KUKA KRL program: f1_Kuka_APT213T03S13.SRC

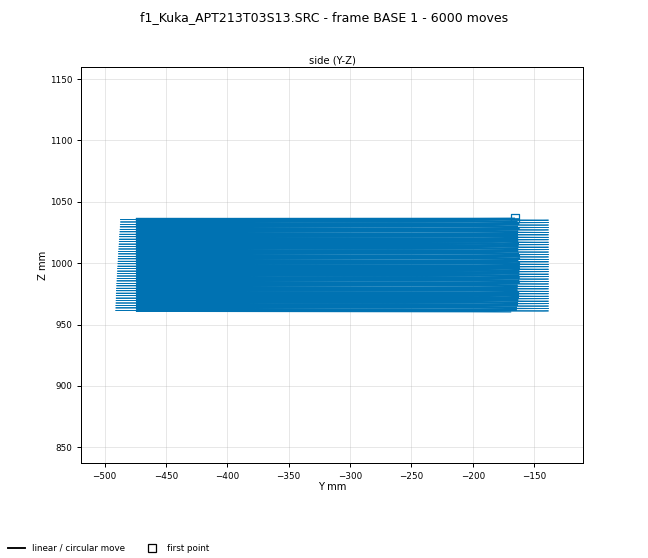
[picture p0: tool path of f1_Kuka_APT213T03S13.SRC in frame BASE 1, 6000 of 6001 moves have a stored position in this frame; points joined in program order, loops and branches not executed]
&ACCESS RVP
&REL 2
&PARAM TEMPLATE = C:\KRC\Roboter\Template\vorgabe
&PARAM EDITMASK = *
DEF f1_Kuka_APT213T03S13()


;FOLD INI;%{PE}%V3.2.0,%MKUKATPBASIS,%CINIT,%VCOMMON,%P
  ;FOLD BAS INI;%{E}%V3.2.0,%MKUKATPBASIS,%CINIT,%VINIT,%P
    GLOBAL INTERRUPT DECL 3 WHEN $STOPMESS==TRUE DO IR_STOPM ( )
    INTERRUPT ON 3
    BAS (#INITMOV,0 )
  ;ENDFOLD (BAS INI)
  ;FOLD USER INI;%{E}%V3.2.0,%MKUKATPUSER,%CINIT,%VINIT,%P
    ;Make your modifications here
  ;ENDFOLD (USER INI)
;ENDFOLD (INI)


;*** Make Null PTP Move
  PTP $pos_act

;*** Auto Load The Correct TOOL Data
  $tool=tool_data[3]

;*** Auto Load The Correct BASE Data
  $base=base_data[1]

  $ADVANCE = 5

;*** Restate Last Velocity
MMPM(30000.0)
SetRPM(6000)
LIN {X 0.063,Y -165.933,Z 1036.809,A 0.000,B 0.000,C 90.000,E1 145.515} C_DIS
LIN {X -0.044,Y -170.922,Z 1036.789,A 0.000,B 0.000,C 90.000,E1 142.065} C_DIS
LIN {X -0.018,Y -175.791,Z 1036.770,A 0.000,B 0.000,C 90.000,E1 138.609} C_DIS
LIN {X -0.018,Y -181.399,Z 1036.751,A 0.000,B 0.000,C 90.000,E1 135.202} C_DIS
LIN {X -0.014,Y -186.897,Z 1036.732,A 0.000,B 0.000,C 90.000,E1 131.838} C_DIS
LIN {X -0.063,Y -191.479,Z 1036.719,A 0.000,B 0.000,C 90.000,E1 129.358} C_DIS
LIN {X -0.019,Y -197.520,Z 1036.700,A 0.000,B 0.000,C 90.000,E1 125.964} C_DIS
LIN {X 0.097,Y -303.588,Z 1036.700,A 0.000,B 0.000,C 90.000,E1 125.931} C_DIS
LIN {X -0.058,Y -305.059,Z 1036.700,A 0.000,B 0.000,C 90.000,E1 125.931} C_DIS
LIN {X 0.134,Y -308.841,Z 1036.699,A 0.000,B 0.000,C 90.000,E1 125.724} C_DIS
LIN {X -0.104,Y -311.070,Z 1036.698,A 0.000,B 0.000,C 90.000,E1 125.598} C_DIS
LIN {X 0.033,Y -314.160,Z 1036.696,A 0.000,B 0.000,C 90.000,E1 125.231} C_DIS
LIN {X -0.057,Y -316.144,Z 1036.694,A 0.000,B 0.000,C 90.000,E1 124.945} C_DIS
LIN {X 0.113,Y -317.699,Z 1036.692,A 0.000,B 0.000,C 90.000,E1 124.612} C_DIS
LIN {X -0.083,Y -319.007,Z 1036.691,A 0.000,B 0.000,C 90.000,E1 124.326} C_DIS
LIN {X -0.008,Y -330.156,Z 1036.673,A 0.000,B 0.000,C 90.000,E1 121.131} C_DIS
LIN {X 0.067,Y -341.560,Z 1036.657,A 0.000,B 0.000,C 90.000,E1 118.309} C_DIS
LIN {X -0.156,Y -354.382,Z 1036.642,A 0.000,B 0.000,C 90.000,E1 115.591} C_DIS
LIN {X 0.094,Y -367.068,Z 1036.629,A 0.000,B 0.000,C 90.000,E1 113.153} C_DIS
LIN {X 0.194,Y -381.055,Z 1036.616,A 0.000,B 0.000,C 90.000,E1 110.791} C_DIS
LIN {X -0.133,Y -396.444,Z 1036.603,A 0.000,B 0.000,C 90.000,E1 108.544} C_DIS
LIN {X 0.173,Y -413.344,Z 1036.590,A 0.000,B 0.000,C 90.000,E1 106.260} C_DIS
LIN {X -0.136,Y -431.875,Z 1036.578,A 0.000,B 0.000,C 90.000,E1 104.120} C_DIS
LIN {X 0.111,Y -451.748,Z 1036.567,A 0.000,B 0.000,C 90.000,E1 102.007} C_DIS
LIN {X 0.212,Y -467.042,Z 1036.559,A 0.000,B 0.000,C 90.000,E1 100.546} C_DIS
LIN {X 0.229,Y -469.174,Z 1036.557,A 0.000,B 0.000,C 90.000,E1 100.310} C_DIS
LIN {X 0.077,Y -470.911,Z 1036.556,A 0.000,B 0.000,C 90.000,E1 100.074} C_DIS
LIN {X -0.158,Y -472.215,Z 1036.555,A 0.000,B 0.000,C 90.000,E1 99.849} C_DIS
LIN {X 0.023,Y -473.839,Z 1036.552,A 0.000,B 0.000,C 90.000,E1 99.321} C_DIS
LIN {X 0.135,Y -474.404,Z 1036.549,A 0.000,B 0.000,C 90.000,E1 98.803} C_DIS
LIN {X -0.211,Y -474.005,Z 1036.546,A 0.000,B 0.000,C 90.000,E1 98.341} C_DIS
LIN {X -0.017,Y -472.586,Z 1036.543,A 0.000,B 0.000,C 90.000,E1 97.814} C_DIS
LIN {X -0.220,Y -471.422,Z 1036.542,A 0.000,B 0.000,C 90.000,E1 97.587} C_DIS
LIN {X -0.100,Y -468.092,Z 1036.539,A 0.000,B 0.000,C 90.000,E1 97.068} C_DIS
LIN {X -0.038,Y -455.730,Z 1036.529,A 0.000,B 0.000,C 90.000,E1 95.277} C_DIS
LIN {X -0.181,Y -438.069,Z 1036.515,A 0.000,B 0.000,C 90.000,E1 92.694} C_DIS
LIN {X -0.168,Y -419.039,Z 1036.497,A 0.000,B 0.000,C 90.000,E1 89.484} C_DIS
LIN {X 0.171,Y -407.384,Z 1036.485,A 0.000,B 0.000,C 90.000,E1 87.249} C_DIS
LIN {X -0.201,Y -396.986,Z 1036.474,A 0.000,B 0.000,C 90.000,E1 85.355} C_DIS
LIN {X 0.031,Y -387.808,Z 1036.465,A 0.000,B 0.000,C 90.000,E1 83.628} C_DIS
LIN {X 0.138,Y -378.455,Z 1036.455,A 0.000,B 0.000,C 90.000,E1 81.894} C_DIS
LIN {X 0.131,Y -368.748,Z 1036.445,A 0.000,B 0.000,C 90.000,E1 80.151} C_DIS
LIN {X -0.087,Y -357.143,Z 1036.434,A 0.000,B 0.000,C 90.000,E1 78.117} C_DIS
LIN {X 0.011,Y -347.219,Z 1036.424,A 0.000,B 0.000,C 90.000,E1 76.297} C_DIS
LIN {X -0.112,Y -334.181,Z 1036.410,A 0.000,B 0.000,C 90.000,E1 73.866} C_DIS
LIN {X 0.058,Y -321.599,Z 1036.396,A 0.000,B 0.000,C 90.000,E1 71.329} C_DIS
LIN {X 0.143,Y -306.483,Z 1036.379,A 0.000,B 0.000,C 90.000,E1 68.103} C_DIS
LIN {X -0.076,Y -296.232,Z 1036.366,A 0.000,B 0.000,C 90.000,E1 65.845} C_DIS
LIN {X 0.120,Y -284.774,Z 1036.351,A 0.000,B 0.000,C 90.000,E1 63.127} C_DIS
LIN {X -0.163,Y -274.969,Z 1036.338,A 0.000,B 0.000,C 90.000,E1 60.795} C_DIS
LIN {X -0.094,Y -263.959,Z 1036.322,A 0.000,B 0.000,C 90.000,E1 57.995} C_DIS
LIN {X 0.116,Y -253.213,Z 1036.306,A 0.000,B 0.000,C 90.000,E1 55.102} C_DIS
LIN {X 0.128,Y -241.650,Z 1036.288,A 0.000,B 0.000,C 90.000,E1 51.823} C_DIS
LIN {X 0.082,Y -230.864,Z 1036.270,A 0.000,B 0.000,C 90.000,E1 48.485} C_DIS
LIN {X -0.075,Y -221.890,Z 1036.253,A 0.000,B 0.000,C 90.000,E1 45.486} C_DIS
LIN {X 0.039,Y -213.400,Z 1036.235,A 0.000,B 0.000,C 90.000,E1 42.366} C_DIS
LIN {X 0.129,Y -205.412,Z 1036.218,A 0.000,B 0.000,C 90.000,E1 39.197} C_DIS
LIN {X 0.081,Y -197.949,Z 1036.200,A 0.000,B 0.000,C 90.000,E1 36.011} C_DIS
LIN {X 0.101,Y -191.076,Z 1036.182,A 0.000,B 0.000,C 90.000,E1 32.752} C_DIS
LIN {X 0.069,Y -184.943,Z 1036.164,A 0.000,B 0.000,C 90.000,E1 29.461} C_DIS
LIN {X -0.060,Y -179.566,Z 1036.145,A 0.000,B 0.000,C 90.000,E1 26.155} C_DIS
LIN {X -0.062,Y -175.003,Z 1036.126,A 0.000,B 0.000,C 90.000,E1 22.770} C_DIS
LIN {X 0.014,Y -171.158,Z 1036.107,A 0.000,B 0.000,C 90.000,E1 19.322} C_DIS
LIN {X -0.003,Y -167.410,Z 1036.083,A 0.000,B 0.000,C 90.000,E1 15.009} C_DIS
LIN {X -0.019,Y -164.696,Z 1036.059,A 0.000,B 0.000,C 90.000,E1 10.658} C_DIS
LIN {X 0.058,Y -162.489,Z 1036.020,A 0.000,B 0.000,C 90.000,E1 3.612} C_DIS
LIN {X -0.061,Y -163.809,Z 1035.963,A 0.000,B 0.000,C 90.000,E1 353.394} C_DIS
LIN {X -0.005,Y -166.537,Z 1035.934,A 0.000,B 0.000,C 90.000,E1 348.117} C_DIS
LIN {X 0.070,Y -169.974,Z 1035.910,A 0.000,B 0.000,C 90.000,E1 343.740} C_DIS
LIN {X -0.022,Y -173.413,Z 1035.891,A 0.000,B 0.000,C 90.000,E1 340.315} C_DIS
LIN {X 0.038,Y -177.583,Z 1035.872,A 0.000,B 0.000,C 90.000,E1 336.869} C_DIS
LIN {X -0.075,Y -182.601,Z 1035.853,A 0.000,B 0.000,C 90.000,E1 333.512} C_DIS
LIN {X 0.025,Y -188.479,Z 1035.834,A 0.000,B 0.000,C 90.000,E1 330.127} C_DIS
LIN {X -0.025,Y -195.149,Z 1035.816,A 0.000,B 0.000,C 90.000,E1 326.834} C_DIS
LIN {X -0.029,Y -202.523,Z 1035.798,A 0.000,B 0.000,C 90.000,E1 323.577} C_DIS
LIN {X 0.034,Y -210.397,Z 1035.780,A 0.000,B 0.000,C 90.000,E1 320.356} C_DIS
LIN {X 0.035,Y -220.038,Z 1035.760,A 0.000,B 0.000,C 90.000,E1 316.824} C_DIS
LIN {X -0.120,Y -229.416,Z 1035.743,A 0.000,B 0.000,C 90.000,E1 313.785} C_DIS
LIN {X -0.158,Y -238.562,Z 1035.728,A 0.000,B 0.000,C 90.000,E1 311.148} C_DIS
LIN {X -0.114,Y -247.580,Z 1035.716,A 0.000,B 0.000,C 90.000,E1 308.910} C_DIS
LIN {X -0.070,Y -256.075,Z 1035.706,A 0.000,B 0.000,C 90.000,E1 307.076} C_DIS
LIN {X 0.008,Y -265.532,Z 1035.696,A 0.000,B 0.000,C 90.000,E1 305.264} C_DIS
LIN {X -0.056,Y -283.955,Z 1035.678,A 0.000,B 0.000,C 90.000,E1 302.133} C_DIS
LIN {X 0.043,Y -303.913,Z 1035.662,A 0.000,B 0.000,C 90.000,E1 299.077} C_DIS
LIN {X 0.026,Y -320.653,Z 1035.649,A 0.000,B 0.000,C 90.000,E1 296.796} C_DIS
LIN {X 0.026,Y -333.786,Z 1035.640,A 0.000,B 0.000,C 90.000,E1 295.207} C_DIS
LIN {X 0.005,Y -350.088,Z 1035.630,A 0.000,B 0.000,C 90.000,E1 293.462} C_DIS
LIN {X 0.000,Y -374.980,Z 1035.617,A 0.000,B 0.000,C 90.000,E1 291.099} C_DIS
LIN {X -0.066,Y -388.784,Z 1035.610,A 0.000,B 0.000,C 90.000,E1 289.885} C_DIS
LIN {X -0.057,Y -402.518,Z 1035.604,A 0.000,B 0.000,C 90.000,E1 288.671} C_DIS
LIN {X 0.025,Y -413.232,Z 1035.598,A 0.000,B 0.000,C 90.000,E1 287.692} C_DIS
LIN {X -0.064,Y -420.992,Z 1035.594,A 0.000,B 0.000,C 90.000,E1 286.968} C_DIS
LIN {X -0.093,Y -428.488,Z 1035.590,A 0.000,B 0.000,C 90.000,E1 286.205} C_DIS
LIN {X 0.073,Y -438.206,Z 1035.584,A 0.000,B 0.000,C 90.000,E1 285.134} C_DIS
LIN {X 0.162,Y -447.427,Z 1035.578,A 0.000,B 0.000,C 90.000,E1 284.064} C_DIS
LIN {X -0.004,Y -453.748,Z 1035.574,A 0.000,B 0.000,C 90.000,E1 283.300} C_DIS
LIN {X -0.110,Y -459.574,Z 1035.570,A 0.000,B 0.000,C 90.000,E1 282.535} C_DIS
LIN {X -0.173,Y -464.897,Z 1035.565,A 0.000,B 0.000,C 90.000,E1 281.771} C_DIS
LIN {X -0.187,Y -469.646,Z 1035.561,A 0.000,B 0.000,C 90.000,E1 281.007} C_DIS
LIN {X 0.212,Y -473.791,Z 1035.557,A 0.000,B 0.000,C 90.000,E1 280.197} C_DIS
LIN {X 0.195,Y -477.338,Z 1035.553,A 0.000,B 0.000,C 90.000,E1 279.443} C_DIS
LIN {X -0.268,Y -480.332,Z 1035.548,A 0.000,B 0.000,C 90.000,E1 278.746} C_DIS
LIN {X -0.047,Y -482.023,Z 1035.546,A 0.000,B 0.000,C 90.000,E1 278.219} C_DIS
LIN {X -0.190,Y -484.661,Z 1035.540,A 0.000,B 0.000,C 90.000,E1 277.239} C_DIS
LIN {X -0.007,Y -485.661,Z 1035.537,A 0.000,B 0.000,C 90.000,E1 276.720} C_DIS
LIN {X 0.186,Y -486.404,Z 1035.535,A 0.000,B 0.000,C 90.000,E1 276.201} C_DIS
LIN {X -0.101,Y -486.901,Z 1035.532,A 0.000,B 0.000,C 90.000,E1 275.739} C_DIS
LIN {X 0.100,Y -487.025,Z 1035.529,A 0.000,B 0.000,C 90.000,E1 275.220} C_DIS
LIN {X -0.183,Y -486.708,Z 1035.526,A 0.000,B 0.000,C 90.000,E1 274.759} C_DIS
LIN {X -0.019,Y -485.861,Z 1035.524,A 0.000,B 0.000,C 90.000,E1 274.245} C_DIS
LIN {X 0.180,Y -484.498,Z 1035.521,A 0.000,B 0.000,C 90.000,E1 273.726} C_DIS
LIN {X -0.141,Y -482.530,Z 1035.518,A 0.000,B 0.000,C 90.000,E1 273.269} C_DIS
LIN {X 0.204,Y -481.280,Z 1035.517,A 0.000,B 0.000,C 90.000,E1 272.980} C_DIS
LIN {X -0.129,Y -478.168,Z 1035.514,A 0.000,B 0.000,C 90.000,E1 272.522} C_DIS
LIN {X 0.002,Y -474.277,Z 1035.511,A 0.000,B 0.000,C 90.000,E1 272.007} C_DIS
LIN {X 0.126,Y -469.504,Z 1035.508,A 0.000,B 0.000,C 90.000,E1 271.489} C_DIS
LIN {X -0.108,Y -464.065,Z 1035.506,A 0.000,B 0.000,C 90.000,E1 271.031} C_DIS
LIN {X -0.020,Y -458.141,Z 1035.503,A 0.000,B 0.000,C 90.000,E1 270.573} C_DIS
LIN {X 0.113,Y -454.937,Z 1035.502,A 0.000,B 0.000,C 90.000,E1 270.344} C_DIS
LIN {X -0.132,Y -448.182,Z 1035.500,A 0.000,B 0.000,C 90.000,E1 270.000} C_DIS
LIN {X 0.097,Y -440.660,Z 1035.498,A 0.000,B 0.000,C 90.000,E1 269.656} C_DIS
LIN {X 0.026,Y -432.481,Z 1035.497,A 0.000,B 0.000,C 90.000,E1 269.427} C_DIS
LIN {X 0.074,Y -423.893,Z 1035.496,A 0.000,B 0.000,C 90.000,E1 269.255} C_DIS
LIN {X 0.081,Y -414.964,Z 1035.495,A 0.000,B 0.000,C 90.000,E1 269.141} C_DIS
LIN {X 0.181,Y -401.514,Z 1035.495,A 0.000,B 0.000,C 90.000,E1 269.026} C_DIS
LIN {X 0.067,Y -397.775,Z 1035.495,A 0.000,B 0.000,C 90.000,E1 269.026} C_DIS
LIN {X 0.005,Y -181.325,Z 1035.495,A 0.000,B 0.000,C 90.000,E1 269.026} C_DIS
LIN {X 0.010,Y -180.904,Z 1035.474,A 0.000,B 0.000,C 90.000,E1 265.298} C_DIS
LIN {X -0.041,Y -180.245,Z 1035.464,A 0.000,B 0.000,C 90.000,E1 263.628} C_DIS
LIN {X -0.021,Y -178.733,Z 1035.441,A 0.000,B 0.000,C 90.000,E1 259.398} C_DIS
LIN {X 0.046,Y -175.781,Z 1035.413,A 0.000,B 0.000,C 90.000,E1 254.283} C_DIS
LIN {X 0.033,Y -171.965,Z 1035.384,A 0.000,B 0.000,C 90.000,E1 249.156} C_DIS
LIN {X 0.071,Y -171.362,Z 1035.380,A 0.000,B 0.000,C 90.000,E1 248.284} C_DIS
LIN {X 0.048,Y -167.610,Z 1035.355,A 0.000,B 0.000,C 90.000,E1 243.973} C_DIS
LIN {X 0.060,Y -166.258,Z 1035.346,A 0.000,B 0.000,C 90.000,E1 242.231} C_DIS
LIN {X 0.048,Y -163.012,Z 1035.326,A 0.000,B 0.000,C 90.000,E1 238.742} C_DIS
LIN {X -0.040,Y -160.935,Z 1035.312,A 0.000,B 0.000,C 90.000,E1 236.135} C_DIS
LIN {X 0.071,Y -157.694,Z 1035.292,A 0.000,B 0.000,C 90.000,E1 232.557} C_DIS
LIN {X 0.008,Y -155.734,Z 1035.277,A 0.000,B 0.000,C 90.000,E1 229.908} C_DIS
LIN {X 0.062,Y -151.993,Z 1035.252,A 0.000,B 0.000,C 90.000,E1 225.405} C_DIS
LIN {X 0.078,Y -150.237,Z 1035.237,A 0.000,B 0.000,C 90.000,E1 222.690} C_DIS
LIN {X 0.001,Y -146.996,Z 1035.212,A 0.000,B 0.000,C 90.000,E1 218.177} C_DIS
LIN {X -0.009,Y -145.582,Z 1035.197,A 0.000,B 0.000,C 90.000,E1 215.438} C_DIS
LIN {X -0.015,Y -142.971,Z 1035.171,A 0.000,B 0.000,C 90.000,E1 210.846} C_DIS
LIN {X 0.038,Y -141.597,Z 1035.151,A 0.000,B 0.000,C 90.000,E1 207.129} C_DIS
LIN {X -0.046,Y -139.422,Z 1035.115,A 0.000,B 0.000,C 90.000,E1 200.663} C_DIS
LIN {X 0.005,Y -139.149,Z 1035.104,A 0.000,B 0.000,C 90.000,E1 198.779} C_DIS
LIN {X 0.027,Y -138.345,Z 1035.058,A 0.000,B 0.000,C 90.000,E1 190.366} C_DIS
LIN {X 0.013,Y -139.487,Z 1035.006,A 0.000,B 0.000,C 90.000,E1 181.031} C_DIS
LIN {X -0.047,Y -141.088,Z 1034.975,A 0.000,B 0.000,C 90.000,E1 175.469} C_DIS
LIN {X 0.048,Y -142.464,Z 1034.959,A 0.000,B 0.000,C 90.000,E1 172.648} C_DIS
LIN {X -0.004,Y -144.709,Z 1034.934,A 0.000,B 0.000,C 90.000,E1 168.049} C_DIS
LIN {X -0.053,Y -147.307,Z 1034.913,A 0.000,B 0.000,C 90.000,E1 164.393} C_DIS
LIN {X -0.038,Y -150.628,Z 1034.888,A 0.000,B 0.000,C 90.000,E1 159.826} C_DIS
LIN {X 0.039,Y -154.104,Z 1034.868,A 0.000,B 0.000,C 90.000,E1 156.177} C_DIS
LIN {X -0.038,Y -157.528,Z 1034.848,A 0.000,B 0.000,C 90.000,E1 152.615} C_DIS
LIN {X -0.093,Y -161.762,Z 1034.828,A 0.000,B 0.000,C 90.000,E1 149.076} C_DIS
LIN {X 0.012,Y -165.955,Z 1034.808,A 0.000,B 0.000,C 90.000,E1 145.515} C_DIS
LIN {X 0.008,Y -170.948,Z 1034.789,A 0.000,B 0.000,C 90.000,E1 142.029} C_DIS
LIN {X -0.071,Y -175.817,Z 1034.770,A 0.000,B 0.000,C 90.000,E1 138.609} C_DIS
LIN {X 0.056,Y -181.424,Z 1034.751,A 0.000,B 0.000,C 90.000,E1 135.162} C_DIS
LIN {X -0.069,Y -186.927,Z 1034.732,A 0.000,B 0.000,C 90.000,E1 131.838} C_DIS
LIN {X 0.004,Y -191.506,Z 1034.719,A 0.000,B 0.000,C 90.000,E1 129.322} C_DIS
LIN {X -0.039,Y -197.441,Z 1034.700,A 0.000,B 0.000,C 90.000,E1 126.011} C_DIS
LIN {X -0.113,Y -303.232,Z 1034.700,A 0.000,B 0.000,C 90.000,E1 126.011} C_DIS
LIN {X 0.026,Y -304.438,Z 1034.700,A 0.000,B 0.000,C 90.000,E1 125.964} C_DIS
LIN {X -0.118,Y -308.771,Z 1034.699,A 0.000,B 0.000,C 90.000,E1 125.804} C_DIS
LIN {X -0.014,Y -311.160,Z 1034.698,A 0.000,B 0.000,C 90.000,E1 125.598} C_DIS
LIN {X -0.056,Y -314.414,Z 1034.696,A 0.000,B 0.000,C 90.000,E1 125.231} C_DIS
LIN {X 0.063,Y -316.358,Z 1034.694,A 0.000,B 0.000,C 90.000,E1 124.898} C_DIS
LIN {X -0.076,Y -317.878,Z 1034.692,A 0.000,B 0.000,C 90.000,E1 124.612} C_DIS
LIN {X -0.205,Y -320.168,Z 1034.689,A 0.000,B 0.000,C 90.000,E1 123.992} C_DIS
LIN {X 0.082,Y -330.261,Z 1034.673,A 0.000,B 0.000,C 90.000,E1 121.082} C_DIS
LIN {X 0.033,Y -341.681,Z 1034.657,A 0.000,B 0.000,C 90.000,E1 118.281} C_DIS
LIN {X -0.037,Y -354.521,Z 1034.642,A 0.000,B 0.000,C 90.000,E1 115.540} C_DIS
LIN {X 0.034,Y -367.223,Z 1034.629,A 0.000,B 0.000,C 90.000,E1 113.131} C_DIS
LIN {X -0.013,Y -381.228,Z 1034.615,A 0.000,B 0.000,C 90.000,E1 110.791} C_DIS
LIN {X 0.031,Y -396.636,Z 1034.603,A 0.000,B 0.000,C 90.000,E1 108.489} C_DIS
LIN {X -0.042,Y -413.556,Z 1034.590,A 0.000,B 0.000,C 90.000,E1 106.260} C_DIS
LIN {X 0.063,Y -432.111,Z 1034.578,A 0.000,B 0.000,C 90.000,E1 104.064} C_DIS
LIN {X -0.102,Y -451.993,Z 1034.567,A 0.000,B 0.000,C 90.000,E1 102.007} C_DIS
LIN {X 0.005,Y -467.278,Z 1034.559,A 0.000,B 0.000,C 90.000,E1 100.546} C_DIS
LIN {X 0.023,Y -469.348,Z 1034.557,A 0.000,B 0.000,C 90.000,E1 100.310} C_DIS
LIN {X -0.129,Y -471.041,Z 1034.556,A 0.000,B 0.000,C 90.000,E1 100.074} C_DIS
LIN {X 0.102,Y -472.311,Z 1034.554,A 0.000,B 0.000,C 90.000,E1 99.792} C_DIS
LIN {X -0.184,Y -473.883,Z 1034.552,A 0.000,B 0.000,C 90.000,E1 99.321} C_DIS
LIN {X -0.071,Y -474.405,Z 1034.549,A 0.000,B 0.000,C 90.000,E1 98.803} C_DIS
LIN {X 0.121,Y -473.964,Z 1034.546,A 0.000,B 0.000,C 90.000,E1 98.276} C_DIS
LIN {X 0.246,Y -472.496,Z 1034.543,A 0.000,B 0.000,C 90.000,E1 97.757} C_DIS
LIN {X 0.042,Y -471.302,Z 1034.542,A 0.000,B 0.000,C 90.000,E1 97.530} C_DIS
LIN {X 0.161,Y -467.931,Z 1034.539,A 0.000,B 0.000,C 90.000,E1 97.011} C_DIS
LIN {X 0.214,Y -455.569,Z 1034.529,A 0.000,B 0.000,C 90.000,E1 95.220} C_DIS
LIN {X 0.059,Y -437.914,Z 1034.515,A 0.000,B 0.000,C 90.000,E1 92.636} C_DIS
LIN {X -0.059,Y -420.406,Z 1034.498,A 0.000,B 0.000,C 90.000,E1 89.714} C_DIS
LIN {X -0.098,Y -408.705,Z 1034.486,A 0.000,B 0.000,C 90.000,E1 87.535} C_DIS
LIN {X -0.031,Y -398.335,Z 1034.475,A 0.000,B 0.000,C 90.000,E1 85.584} C_DIS
LIN {X 0.173,Y -390.772,Z 1034.468,A 0.000,B 0.000,C 90.000,E1 84.147} C_DIS
LIN {X -0.069,Y -379.880,Z 1034.457,A 0.000,B 0.000,C 90.000,E1 82.186} C_DIS
LIN {X -0.053,Y -371.896,Z 1034.448,A 0.000,B 0.000,C 90.000,E1 80.735} C_DIS
LIN {X -0.200,Y -360.299,Z 1034.437,A 0.000,B 0.000,C 90.000,E1 78.701} C_DIS
LIN {X -0.103,Y -348.719,Z 1034.425,A 0.000,B 0.000,C 90.000,E1 76.589} C_DIS
LIN {X 0.139,Y -335.665,Z 1034.412,A 0.000,B 0.000,C 90.000,E1 74.102} C_DIS
LIN {X -0.070,Y -323.026,Z 1034.398,A 0.000,B 0.000,C 90.000,E1 71.638} C_DIS
LIN {X 0.062,Y -307.822,Z 1034.380,A 0.000,B 0.000,C 90.000,E1 68.411} C_DIS
LIN {X 0.030,Y -296.106,Z 1034.366,A 0.000,B 0.000,C 90.000,E1 65.793} C_DIS
LIN {X -0.041,Y -284.638,Z 1034.351,A 0.000,B 0.000,C 90.000,E1 63.127} C_DIS
LIN {X 0.052,Y -274.820,Z 1034.337,A 0.000,B 0.000,C 90.000,E1 60.717} C_DIS
LIN {X 0.114,Y -263.802,Z 1034.322,A 0.000,B 0.000,C 90.000,E1 57.916} C_DIS
LIN {X -0.013,Y -251.723,Z 1034.304,A 0.000,B 0.000,C 90.000,E1 54.736} C_DIS
LIN {X -0.027,Y -240.271,Z 1034.286,A 0.000,B 0.000,C 90.000,E1 51.457} C_DIS
LIN {X 0.042,Y -229.561,Z 1034.267,A 0.000,B 0.000,C 90.000,E1 48.081} C_DIS
LIN {X -0.059,Y -219.588,Z 1034.248,A 0.000,B 0.000,C 90.000,E1 44.676} C_DIS
LIN {X 0.015,Y -211.170,Z 1034.231,A 0.000,B 0.000,C 90.000,E1 41.553} C_DIS
LIN {X 0.054,Y -203.300,Z 1034.213,A 0.000,B 0.000,C 90.000,E1 38.382} C_DIS
LIN {X -0.001,Y -195.952,Z 1034.195,A 0.000,B 0.000,C 90.000,E1 35.185} C_DIS
LIN {X -0.024,Y -189.285,Z 1034.177,A 0.000,B 0.000,C 90.000,E1 31.926} C_DIS
LIN {X -0.031,Y -183.335,Z 1034.159,A 0.000,B 0.000,C 90.000,E1 28.615} C_DIS
LIN {X -0.112,Y -178.162,Z 1034.140,A 0.000,B 0.000,C 90.000,E1 25.283} C_DIS
LIN {X 0.018,Y -173.827,Z 1034.121,A 0.000,B 0.000,C 90.000,E1 21.844} C_DIS
LIN {X 0.004,Y -170.155,Z 1034.102,A 0.000,B 0.000,C 90.000,E1 18.417} C_DIS
LIN {X 0.072,Y -166.653,Z 1034.078,A 0.000,B 0.000,C 90.000,E1 14.064} C_DIS
LIN {X -0.027,Y -163.790,Z 1034.049,A 0.000,B 0.000,C 90.000,E1 8.859} C_DIS
LIN {X 0.038,Y -164.476,Z 1033.953,A 0.000,B 0.000,C 90.000,E1 351.602} C_DIS
LIN {X 0.046,Y -167.694,Z 1033.924,A 0.000,B 0.000,C 90.000,E1 346.353} C_DIS
LIN {X 0.088,Y -171.524,Z 1033.900,A 0.000,B 0.000,C 90.000,E1 342.000} C_DIS
LIN {X -0.016,Y -175.313,Z 1033.881,A 0.000,B 0.000,C 90.000,E1 338.592} C_DIS
LIN {X -0.003,Y -179.939,Z 1033.862,A 0.000,B 0.000,C 90.000,E1 335.177} C_DIS
LIN {X 0.105,Y -185.373,Z 1033.843,A 0.000,B 0.000,C 90.000,E1 331.769} C_DIS
LIN {X 0.045,Y -191.674,Z 1033.825,A 0.000,B 0.000,C 90.000,E1 328.456} C_DIS
LIN {X 0.014,Y -198.736,Z 1033.807,A 0.000,B 0.000,C 90.000,E1 325.182} C_DIS
LIN {X 0.060,Y -207.325,Z 1033.786,A 0.000,B 0.000,C 90.000,E1 321.537} C_DIS
LIN {X -0.062,Y -215.614,Z 1033.769,A 0.000,B 0.000,C 90.000,E1 318.405} C_DIS
LIN {X -0.094,Y -225.706,Z 1033.749,A 0.000,B 0.000,C 90.000,E1 314.919} C_DIS
LIN {X 0.064,Y -235.779,Z 1033.733,A 0.000,B 0.000,C 90.000,E1 311.838} C_DIS
LIN {X -0.088,Y -241.394,Z 1033.724,A 0.000,B 0.000,C 90.000,E1 310.378} C_DIS
LIN {X -0.144,Y -250.806,Z 1033.712,A 0.000,B 0.000,C 90.000,E1 308.177} C_DIS
LIN {X 0.158,Y -259.687,Z 1033.702,A 0.000,B 0.000,C 90.000,E1 306.297} C_DIS
LIN {X -0.005,Y -275.563,Z 1033.686,A 0.000,B 0.000,C 90.000,E1 303.499} C_DIS
LIN {X -0.001,Y -294.838,Z 1033.669,A 0.000,B 0.000,C 90.000,E1 300.413} C_DIS
LIN {X 0.016,Y -315.797,Z 1033.652,A 0.000,B 0.000,C 90.000,E1 297.436} C_DIS
LIN {X -0.083,Y -328.551,Z 1033.644,A 0.000,B 0.000,C 90.000,E1 295.848} C_DIS
LIN {X -0.081,Y -344.883,Z 1033.633,A 0.000,B 0.000,C 90.000,E1 294.027} C_DIS
LIN {X -0.141,Y -372.528,Z 1033.619,A 0.000,B 0.000,C 90.000,E1 291.354} C_DIS
LIN {X -0.141,Y -386.409,Z 1033.612,A 0.000,B 0.000,C 90.000,E1 290.120} C_DIS
LIN {X -0.109,Y -402.898,Z 1033.604,A 0.000,B 0.000,C 90.000,E1 288.652} C_DIS
LIN {X 0.214,Y -413.603,Z 1033.598,A 0.000,B 0.000,C 90.000,E1 287.638} C_DIS
LIN {X 0.134,Y -421.287,Z 1033.594,A 0.000,B 0.000,C 90.000,E1 286.913} C_DIS
LIN {X -0.017,Y -431.281,Z 1033.588,A 0.000,B 0.000,C 90.000,E1 285.898} C_DIS
LIN {X -0.225,Y -438.537,Z 1033.584,A 0.000,B 0.000,C 90.000,E1 285.134} C_DIS
LIN {X -0.138,Y -447.685,Z 1033.578,A 0.000,B 0.000,C 90.000,E1 284.064} C_DIS
LIN {X 0.136,Y -453.998,Z 1033.574,A 0.000,B 0.000,C 90.000,E1 283.244} C_DIS
LIN {X 0.035,Y -459.820,Z 1033.569,A 0.000,B 0.000,C 90.000,E1 282.479} C_DIS
LIN {X -0.023,Y -465.087,Z 1033.565,A 0.000,B 0.000,C 90.000,E1 281.715} C_DIS
LIN {X -0.033,Y -469.834,Z 1033.561,A 0.000,B 0.000,C 90.000,E1 280.950} C_DIS
LIN {X -0.096,Y -473.977,Z 1033.557,A 0.000,B 0.000,C 90.000,E1 280.197} C_DIS
LIN {X -0.114,Y -477.505,Z 1033.552,A 0.000,B 0.000,C 90.000,E1 279.443} C_DIS
LIN {X -0.030,Y -480.497,Z 1033.548,A 0.000,B 0.000,C 90.000,E1 278.681} C_DIS
LIN {X 0.121,Y -482.174,Z 1033.545,A 0.000,B 0.000,C 90.000,E1 278.163} C_DIS
LIN {X -0.194,Y -483.602,Z 1033.543,A 0.000,B 0.000,C 90.000,E1 277.701} C_DIS
LIN {X -0.018,Y -484.795,Z 1033.540,A 0.000,B 0.000,C 90.000,E1 277.182} C_DIS
LIN {X 0.168,Y -485.781,Z 1033.537,A 0.000,B 0.000,C 90.000,E1 276.663} C_DIS
LIN {X -0.123,Y -486.548,Z 1033.534,A 0.000,B 0.000,C 90.000,E1 276.201} C_DIS
LIN {X 0.075,Y -487.020,Z 1033.532,A 0.000,B 0.000,C 90.000,E1 275.682} C_DIS
LIN {X -0.207,Y -487.112,Z 1033.529,A 0.000,B 0.000,C 90.000,E1 275.220} C_DIS
LIN {X -0.005,Y -486.768,Z 1033.526,A 0.000,B 0.000,C 90.000,E1 274.702} C_DIS
LIN {X 0.159,Y -485.937,Z 1033.523,A 0.000,B 0.000,C 90.000,E1 274.188} C_DIS
LIN {X -0.125,Y -484.522,Z 1033.521,A 0.000,B 0.000,C 90.000,E1 273.726} C_DIS
LIN {X 0.039,Y -482.552,Z 1033.518,A 0.000,B 0.000,C 90.000,E1 273.212} C_DIS
LIN {X -0.098,Y -481.300,Z 1033.516,A 0.000,B 0.000,C 90.000,E1 272.980} C_DIS
LIN {X 0.049,Y -478.133,Z 1033.514,A 0.000,B 0.000,C 90.000,E1 272.465} C_DIS
LIN {X 0.179,Y -474.283,Z 1033.511,A 0.000,B 0.000,C 90.000,E1 271.949} C_DIS
LIN {X -0.168,Y -469.504,Z 1033.508,A 0.000,B 0.000,C 90.000,E1 271.489} C_DIS
LIN {X 0.065,Y -464.001,Z 1033.505,A 0.000,B 0.000,C 90.000,E1 270.974} C_DIS
LIN {X 0.137,Y -458.011,Z 1033.503,A 0.000,B 0.000,C 90.000,E1 270.516} C_DIS
LIN {X 0.170,Y -451.603,Z 1033.501,A 0.000,B 0.000,C 90.000,E1 270.115} C_DIS
LIN {X -0.192,Y -444.672,Z 1033.499,A 0.000,B 0.000,C 90.000,E1 269.828} C_DIS
LIN {X -0.044,Y -437.078,Z 1033.497,A 0.000,B 0.000,C 90.000,E1 269.542} C_DIS
LIN {X 0.163,Y -428.712,Z 1033.496,A 0.000,B 0.000,C 90.000,E1 269.312} C_DIS
LIN {X -0.036,Y -419.953,Z 1033.495,A 0.000,B 0.000,C 90.000,E1 269.198} C_DIS
LIN {X 0.076,Y -410.553,Z 1033.495,A 0.000,B 0.000,C 90.000,E1 269.083} C_DIS
LIN {X -0.040,Y -397.684,Z 1033.495,A 0.000,B 0.000,C 90.000,E1 269.026} C_DIS
LIN {X -0.044,Y -181.321,Z 1033.495,A 0.000,B 0.000,C 90.000,E1 269.026} C_DIS
LIN {X -0.039,Y -180.903,Z 1033.474,A 0.000,B 0.000,C 90.000,E1 265.298} C_DIS
LIN {X -0.089,Y -180.238,Z 1033.464,A 0.000,B 0.000,C 90.000,E1 263.628} C_DIS
LIN {X -0.069,Y -178.724,Z 1033.441,A 0.000,B 0.000,C 90.000,E1 259.398} C_DIS
LIN {X -0.001,Y -175.771,Z 1033.413,A 0.000,B 0.000,C 90.000,E1 254.283} C_DIS
LIN {X -0.013,Y -171.955,Z 1033.384,A 0.000,B 0.000,C 90.000,E1 249.156} C_DIS
LIN {X 0.024,Y -171.347,Z 1033.379,A 0.000,B 0.000,C 90.000,E1 248.284} C_DIS
LIN {X 0.002,Y -167.599,Z 1033.355,A 0.000,B 0.000,C 90.000,E1 243.973} C_DIS
LIN {X 0.014,Y -166.241,Z 1033.346,A 0.000,B 0.000,C 90.000,E1 242.231} C_DIS
LIN {X 0.002,Y -162.999,Z 1033.326,A 0.000,B 0.000,C 90.000,E1 238.742} C_DIS
LIN {X 0.049,Y -160.918,Z 1033.312,A 0.000,B 0.000,C 90.000,E1 236.087} C_DIS
LIN {X 0.027,Y -157.681,Z 1033.292,A 0.000,B 0.000,C 90.000,E1 232.557} C_DIS
LIN {X -0.035,Y -155.721,Z 1033.277,A 0.000,B 0.000,C 90.000,E1 229.908} C_DIS
LIN {X 0.019,Y -151.980,Z 1033.252,A 0.000,B 0.000,C 90.000,E1 225.405} C_DIS
LIN {X 0.036,Y -150.225,Z 1033.237,A 0.000,B 0.000,C 90.000,E1 222.690} C_DIS
LIN {X -0.042,Y -146.987,Z 1033.212,A 0.000,B 0.000,C 90.000,E1 218.177} C_DIS
LIN {X -0.051,Y -145.572,Z 1033.197,A 0.000,B 0.000,C 90.000,E1 215.438} C_DIS
LIN {X 0.067,Y -142.962,Z 1033.171,A 0.000,B 0.000,C 90.000,E1 210.797} C_DIS
LIN {X -0.003,Y -141.589,Z 1033.151,A 0.000,B 0.000,C 90.000,E1 207.129} C_DIS
LIN {X 0.043,Y -139.419,Z 1033.115,A 0.000,B 0.000,C 90.000,E1 200.610} C_DIS
LIN {X -0.036,Y -139.146,Z 1033.104,A 0.000,B 0.000,C 90.000,E1 198.779} C_DIS
LIN {X -0.013,Y -138.347,Z 1033.058,A 0.000,B 0.000,C 90.000,E1 190.366} C_DIS
LIN {X -0.028,Y -139.489,Z 1033.006,A 0.000,B 0.000,C 90.000,E1 181.031} C_DIS
LIN {X 0.052,Y -141.095,Z 1032.975,A 0.000,B 0.000,C 90.000,E1 175.412} C_DIS
LIN {X 0.006,Y -142.473,Z 1032.959,A 0.000,B 0.000,C 90.000,E1 172.648} C_DIS
LIN {X -0.046,Y -144.719,Z 1032.933,A 0.000,B 0.000,C 90.000,E1 168.049} C_DIS
LIN {X 0.047,Y -147.320,Z 1032.913,A 0.000,B 0.000,C 90.000,E1 164.338} C_DIS
LIN {X -0.029,Y -150.642,Z 1032.888,A 0.000,B 0.000,C 90.000,E1 159.806} C_DIS
LIN {X -0.006,Y -154.120,Z 1032.868,A 0.000,B 0.000,C 90.000,E1 156.177} C_DIS
LIN {X -0.082,Y -157.545,Z 1032.848,A 0.000,B 0.000,C 90.000,E1 152.615} C_DIS
LIN {X 0.083,Y -161.784,Z 1032.828,A 0.000,B 0.000,C 90.000,E1 148.997} C_DIS
LIN {X -0.034,Y -165.976,Z 1032.808,A 0.000,B 0.000,C 90.000,E1 145.515} C_DIS
LIN {X -0.038,Y -170.971,Z 1032.789,A 0.000,B 0.000,C 90.000,E1 142.029} C_DIS
LIN {X 0.013,Y -175.840,Z 1032.770,A 0.000,B 0.000,C 90.000,E1 138.566} C_DIS
LIN {X 0.008,Y -181.446,Z 1032.751,A 0.000,B 0.000,C 90.000,E1 135.162} C_DIS
LIN {X -0.119,Y -186.954,Z 1032.732,A 0.000,B 0.000,C 90.000,E1 131.838} C_DIS
LIN {X 0.003,Y -190.067,Z 1032.723,A 0.000,B 0.000,C 90.000,E1 130.135} C_DIS
LIN {X 0.116,Y -197.354,Z 1032.700,A 0.000,B 0.000,C 90.000,E1 126.011} C_DIS
LIN {X 0.118,Y -302.474,Z 1032.700,A 0.000,B 0.000,C 90.000,E1 126.011} C_DIS
LIN {X -0.010,Y -306.647,Z 1032.700,A 0.000,B 0.000,C 90.000,E1 125.931} C_DIS
LIN {X 0.074,Y -309.780,Z 1032.698,A 0.000,B 0.000,C 90.000,E1 125.724} C_DIS
LIN {X -0.128,Y -313.455,Z 1032.697,A 0.000,B 0.000,C 90.000,E1 125.391} C_DIS
LIN {X -0.086,Y -316.965,Z 1032.693,A 0.000,B 0.000,C 90.000,E1 124.818} C_DIS
LIN {X -0.029,Y -318.374,Z 1032.692,A 0.000,B 0.000,C 90.000,E1 124.485} C_DIS
LIN {X -0.143,Y -330.686,Z 1032.672,A 0.000,B 0.000,C 90.000,E1 121.003} C_DIS
LIN {X 0.112,Y -342.160,Z 1032.656,A 0.000,B 0.000,C 90.000,E1 118.153} C_DIS
LIN {X 0.056,Y -355.065,Z 1032.641,A 0.000,B 0.000,C 90.000,E1 115.412} C_DIS
LIN {X -0.002,Y -367.826,Z 1032.628,A 0.000,B 0.000,C 90.000,E1 113.025} C_DIS
LIN {X 0.111,Y -381.894,Z 1032.615,A 0.000,B 0.000,C 90.000,E1 110.663} C_DIS
LIN {X 0.173,Y -397.371,Z 1032.602,A 0.000,B 0.000,C 90.000,E1 108.362} C_DIS
LIN {X 0.117,Y -414.365,Z 1032.590,A 0.000,B 0.000,C 90.000,E1 106.134} C_DIS
LIN {X 0.139,Y -432.998,Z 1032.578,A 0.000,B 0.000,C 90.000,E1 103.953} C_DIS
LIN {X 0.124,Y -452.933,Z 1032.566,A 0.000,B 0.000,C 90.000,E1 101.883} C_DIS
LIN {X 0.196,Y -468.118,Z 1032.558,A 0.000,B 0.000,C 90.000,E1 100.433} C_DIS
LIN {X 0.146,Y -470.038,Z 1032.557,A 0.000,B 0.000,C 90.000,E1 100.197} C_DIS
LIN {X 0.096,Y -471.495,Z 1032.555,A 0.000,B 0.000,C 90.000,E1 99.962} C_DIS
LIN {X 0.193,Y -473.477,Z 1032.553,A 0.000,B 0.000,C 90.000,E1 99.443} C_DIS
LIN {X -0.092,Y -474.336,Z 1032.550,A 0.000,B 0.000,C 90.000,E1 98.973} C_DIS
LIN {X 0.028,Y -474.218,Z 1032.547,A 0.000,B 0.000,C 90.000,E1 98.454} C_DIS
LIN {X 0.155,Y -473.114,Z 1032.544,A 0.000,B 0.000,C 90.000,E1 97.936} C_DIS
LIN {X 0.015,Y -472.141,Z 1032.543,A 0.000,B 0.000,C 90.000,E1 97.701} C_DIS
LIN {X -0.124,Y -470.828,Z 1032.541,A 0.000,B 0.000,C 90.000,E1 97.466} C_DIS
LIN {X -0.068,Y -458.526,Z 1032.531,A 0.000,B 0.000,C 90.000,E1 95.682} C_DIS
LIN {X -0.054,Y -444.216,Z 1032.520,A 0.000,B 0.000,C 90.000,E1 93.612} C_DIS
LIN {X 0.188,Y -429.209,Z 1032.507,A 0.000,B 0.000,C 90.000,E1 91.203} C_DIS
LIN {X 0.117,Y -414.054,Z 1032.492,A 0.000,B 0.000,C 90.000,E1 88.511} C_DIS
LIN {X -0.122,Y -403.801,Z 1032.481,A 0.000,B 0.000,C 90.000,E1 86.617} C_DIS
LIN {X -0.158,Y -393.344,Z 1032.470,A 0.000,B 0.000,C 90.000,E1 84.666} C_DIS
LIN {X 0.035,Y -382.493,Z 1032.459,A 0.000,B 0.000,C 90.000,E1 82.648} C_DIS
LIN {X 0.094,Y -374.584,Z 1032.451,A 0.000,B 0.000,C 90.000,E1 81.197} C_DIS
LIN {X 0.031,Y -366.382,Z 1032.443,A 0.000,B 0.000,C 90.000,E1 79.746} C_DIS
LIN {X -0.162,Y -354.781,Z 1032.432,A 0.000,B 0.000,C 90.000,E1 77.701} C_DIS
LIN {X 0.154,Y -341.626,Z 1032.418,A 0.000,B 0.000,C 90.000,E1 75.227} C_DIS
LIN {X -0.009,Y -328.803,Z 1032.404,A 0.000,B 0.000,C 90.000,E1 72.779} C_DIS
LIN {X 0.032,Y -316.368,Z 1032.390,A 0.000,B 0.000,C 90.000,E1 70.242} C_DIS
LIN {X -0.018,Y -304.389,Z 1032.376,A 0.000,B 0.000,C 90.000,E1 67.667} C_DIS
LIN {X -0.006,Y -294.199,Z 1032.363,A 0.000,B 0.000,C 90.000,E1 65.357} C_DIS
LIN {X 0.004,Y -282.750,Z 1032.348,A 0.000,B 0.000,C 90.000,E1 62.666} C_DIS
LIN {X 0.058,Y -272.973,Z 1032.335,A 0.000,B 0.000,C 90.000,E1 60.255} C_DIS
LIN {X 0.072,Y -261.940,Z 1032.319,A 0.000,B 0.000,C 90.000,E1 57.454} C_DIS
LIN {X 0.016,Y -251.244,Z 1032.303,A 0.000,B 0.000,C 90.000,E1 54.609} C_DIS
LIN {X -0.022,Y -239.836,Z 1032.285,A 0.000,B 0.000,C 90.000,E1 51.331} C_DIS
LIN {X 0.031,Y -229.143,Z 1032.266,A 0.000,B 0.000,C 90.000,E1 47.957} C_DIS
LIN {X -0.012,Y -220.261,Z 1032.250,A 0.000,B 0.000,C 90.000,E1 44.919} C_DIS
LIN {X -0.079,Y -211.788,Z 1032.232,A 0.000,B 0.000,C 90.000,E1 41.838} C_DIS
LIN {X -0.026,Y -203.841,Z 1032.215,A 0.000,B 0.000,C 90.000,E1 38.669} C_DIS
LIN {X 0.049,Y -196.440,Z 1032.197,A 0.000,B 0.000,C 90.000,E1 35.438} C_DIS
LIN {X -0.072,Y -189.701,Z 1032.179,A 0.000,B 0.000,C 90.000,E1 32.212} C_DIS
LIN {X 0.027,Y -183.679,Z 1032.160,A 0.000,B 0.000,C 90.000,E1 28.871} C_DIS
LIN {X -0.049,Y -178.449,Z 1032.142,A 0.000,B 0.000,C 90.000,E1 25.540} C_DIS
LIN {X -0.073,Y -174.056,Z 1032.123,A 0.000,B 0.000,C 90.000,E1 22.153} C_DIS
LIN {X -0.078,Y -170.335,Z 1032.104,A 0.000,B 0.000,C 90.000,E1 18.725} C_DIS
LIN {X 0.045,Y -166.754,Z 1032.080,A 0.000,B 0.000,C 90.000,E1 14.356} C_DIS
LIN {X -0.026,Y -164.193,Z 1032.056,A 0.000,B 0.000,C 90.000,E1 10.018} C_DIS
LIN {X 0.009,Y -162.268,Z 1032.017,A 0.000,B 0.000,C 90.000,E1 2.980} C_DIS
LIN {X -0.067,Y -163.657,Z 1031.963,A 0.000,B 0.000,C 90.000,E1 353.394} C_DIS
LIN {X -0.017,Y -166.410,Z 1031.934,A 0.000,B 0.000,C 90.000,E1 348.117} C_DIS
LIN {X 0.054,Y -169.827,Z 1031.910,A 0.000,B 0.000,C 90.000,E1 343.740} C_DIS
LIN {X 0.016,Y -173.254,Z 1031.891,A 0.000,B 0.000,C 90.000,E1 340.296} C_DIS
LIN {X 0.013,Y -177.454,Z 1031.871,A 0.000,B 0.000,C 90.000,E1 336.869} C_DIS
LIN {X 0.060,Y -182.494,Z 1031.853,A 0.000,B 0.000,C 90.000,E1 333.461} C_DIS
LIN {X -0.006,Y -188.378,Z 1031.834,A 0.000,B 0.000,C 90.000,E1 330.127} C_DIS
LIN {X -0.061,Y -195.079,Z 1031.816,A 0.000,B 0.000,C 90.000,E1 326.834} C_DIS
LIN {X 0.053,Y -202.442,Z 1031.797,A 0.000,B 0.000,C 90.000,E1 323.543} C_DIS
LIN {X -0.118,Y -211.335,Z 1031.778,A 0.000,B 0.000,C 90.000,E1 319.989} C_DIS
LIN {X -0.107,Y -221.077,Z 1031.758,A 0.000,B 0.000,C 90.000,E1 316.458} C_DIS
LIN {X -0.084,Y -230.539,Z 1031.741,A 0.000,B 0.000,C 90.000,E1 313.380} C_DIS
LIN {X 0.088,Y -239.868,Z 1031.726,A 0.000,B 0.000,C 90.000,E1 310.701} C_DIS
LIN {X -0.026,Y -249.109,Z 1031.714,A 0.000,B 0.000,C 90.000,E1 308.508} C_DIS
LIN {X 0.086,Y -257.798,Z 1031.704,A 0.000,B 0.000,C 90.000,E1 306.664} C_DIS
LIN {X 0.028,Y -273.509,Z 1031.688,A 0.000,B 0.000,C 90.000,E1 303.833} C_DIS
LIN {X -0.026,Y -292.655,Z 1031.671,A 0.000,B 0.000,C 90.000,E1 300.747} C_DIS
LIN {X -0.080,Y -313.469,Z 1031.654,A 0.000,B 0.000,C 90.000,E1 297.769} C_DIS
LIN {X -0.064,Y -326.019,Z 1031.645,A 0.000,B 0.000,C 90.000,E1 296.155} C_DIS
LIN {X -0.091,Y -339.253,Z 1031.637,A 0.000,B 0.000,C 90.000,E1 294.643} C_DIS
LIN {X -0.161,Y -355.809,Z 1031.627,A 0.000,B 0.000,C 90.000,E1 292.950} C_DIS
LIN {X -0.025,Y -380.805,Z 1031.615,A 0.000,B 0.000,C 90.000,E1 290.610} C_DIS
LIN {X -0.033,Y -397.334,Z 1031.606,A 0.000,B 0.000,C 90.000,E1 289.141} C_DIS
LIN {X -0.091,Y -410.802,Z 1031.600,A 0.000,B 0.000,C 90.000,E1 287.946} C_DIS
LIN {X -0.147,Y -418.551,Z 1031.596,A 0.000,B 0.000,C 90.000,E1 287.221} C_DIS
LIN {X 0.091,Y -426.006,Z 1031.591,A 0.000,B 0.000,C 90.000,E1 286.441} C_DIS
LIN {X -0.205,Y -435.843,Z 1031.586,A 0.000,B 0.000,C 90.000,E1 285.426} C_DIS
LIN {X 0.071,Y -442.866,Z 1031.581,A 0.000,B 0.000,C 90.000,E1 284.592} C_DIS
LIN {X -0.138,Y -449.533,Z 1031.577,A 0.000,B 0.000,C 90.000,E1 283.828} C_DIS
LIN {X 0.161,Y -455.718,Z 1031.572,A 0.000,B 0.000,C 90.000,E1 283.008} C_DIS
LIN {X 0.070,Y -461.404,Z 1031.568,A 0.000,B 0.000,C 90.000,E1 282.243} C_DIS
LIN {X -0.131,Y -468.142,Z 1031.562,A 0.000,B 0.000,C 90.000,E1 281.243} C_DIS
LIN {X -0.205,Y -472.518,Z 1031.558,A 0.000,B 0.000,C 90.000,E1 280.489} C_DIS
LIN {X -0.161,Y -476.264,Z 1031.554,A 0.000,B 0.000,C 90.000,E1 279.726} C_DIS
LIN {X -0.035,Y -478.477,Z 1031.551,A 0.000,B 0.000,C 90.000,E1 279.208} C_DIS
LIN {X 0.109,Y -480.421,Z 1031.548,A 0.000,B 0.000,C 90.000,E1 278.690} C_DIS
LIN {X -0.144,Y -482.113,Z 1031.546,A 0.000,B 0.000,C 90.000,E1 278.219} C_DIS
LIN {X 0.019,Y -483.575,Z 1031.543,A 0.000,B 0.000,C 90.000,E1 277.701} C_DIS
LIN {X 0.195,Y -484.783,Z 1031.540,A 0.000,B 0.000,C 90.000,E1 277.182} C_DIS
LIN {X -0.102,Y -485.799,Z 1031.537,A 0.000,B 0.000,C 90.000,E1 276.720} C_DIS
LIN {X 0.091,Y -486.599,Z 1031.535,A 0.000,B 0.000,C 90.000,E1 276.201} C_DIS
LIN {X -0.195,Y -487.098,Z 1031.532,A 0.000,B 0.000,C 90.000,E1 275.739} C_DIS
LIN {X 0.006,Y -487.226,Z 1031.529,A 0.000,B 0.000,C 90.000,E1 275.220} C_DIS
LIN {X 0.209,Y -486.918,Z 1031.526,A 0.000,B 0.000,C 90.000,E1 274.702} C_DIS
LIN {X -0.110,Y -486.136,Z 1031.524,A 0.000,B 0.000,C 90.000,E1 274.245} C_DIS
LIN {X 0.091,Y -484.769,Z 1031.521,A 0.000,B 0.000,C 90.000,E1 273.726} C_DIS
LIN {X -0.229,Y -482.840,Z 1031.518,A 0.000,B 0.000,C 90.000,E1 273.269} C_DIS
LIN {X 0.117,Y -481.646,Z 1031.517,A 0.000,B 0.000,C 90.000,E1 272.980} C_DIS
LIN {X -0.213,Y -478.640,Z 1031.514,A 0.000,B 0.000,C 90.000,E1 272.522} C_DIS
LIN {X -0.079,Y -474.808,Z 1031.511,A 0.000,B 0.000,C 90.000,E1 272.007} C_DIS
LIN {X 0.049,Y -470.150,Z 1031.508,A 0.000,B 0.000,C 90.000,E1 271.489} C_DIS
LIN {X -0.213,Y -464.678,Z 1031.506,A 0.000,B 0.000,C 90.000,E1 271.031} C_DIS
LIN {X 0.171,Y -461.729,Z 1031.504,A 0.000,B 0.000,C 90.000,E1 270.745} C_DIS
LIN {X -0.091,Y -455.353,Z 1031.502,A 0.000,B 0.000,C 90.000,E1 270.344} C_DIS
LIN {X 0.147,Y -448.638,Z 1031.500,A 0.000,B 0.000,C 90.000,E1 269.943} C_DIS
LIN {X -0.014,Y -441.321,Z 1031.498,A 0.000,B 0.000,C 90.000,E1 269.656} C_DIS
LIN {X -0.085,Y -433.338,Z 1031.497,A 0.000,B 0.000,C 90.000,E1 269.427} C_DIS
LIN {X -0.087,Y -424.510,Z 1031.496,A 0.000,B 0.000,C 90.000,E1 269.255} C_DIS
LIN {X -0.089,Y -415.613,Z 1031.495,A 0.000,B 0.000,C 90.000,E1 269.141} C_DIS
LIN {X 0.126,Y -405.608,Z 1031.495,A 0.000,B 0.000,C 90.000,E1 269.026} C_DIS
LIN {X -0.166,Y -394.972,Z 1031.495,A 0.000,B 0.000,C 90.000,E1 269.026} C_DIS
LIN {X 0.078,Y -181.317,Z 1031.494,A 0.000,B 0.000,C 90.000,E1 268.969} C_DIS
LIN {X -0.075,Y -180.902,Z 1031.474,A 0.000,B 0.000,C 90.000,E1 265.298} C_DIS
LIN {X 0.055,Y -180.233,Z 1031.464,A 0.000,B 0.000,C 90.000,E1 263.571} C_DIS
LIN {X 0.070,Y -178.716,Z 1031.441,A 0.000,B 0.000,C 90.000,E1 259.342} C_DIS
LIN {X -0.036,Y -175.765,Z 1031.413,A 0.000,B 0.000,C 90.000,E1 254.283} C_DIS
LIN {X 0.013,Y -171.948,Z 1031.384,A 0.000,B 0.000,C 90.000,E1 249.135} C_DIS
LIN {X -0.011,Y -171.336,Z 1031.379,A 0.000,B 0.000,C 90.000,E1 248.284} C_DIS
LIN {X -0.032,Y -167.590,Z 1031.355,A 0.000,B 0.000,C 90.000,E1 243.973} C_DIS
LIN {X -0.020,Y -166.228,Z 1031.346,A 0.000,B 0.000,C 90.000,E1 242.231} C_DIS
LIN {X -0.032,Y -162.989,Z 1031.326,A 0.000,B 0.000,C 90.000,E1 238.742} C_DIS
LIN {X 0.015,Y -160.906,Z 1031.312,A 0.000,B 0.000,C 90.000,E1 236.087} C_DIS
LIN {X -0.007,Y -157.672,Z 1031.292,A 0.000,B 0.000,C 90.000,E1 232.557} C_DIS
LIN {X -0.068,Y -155.710,Z 1031.277,A 0.000,B 0.000,C 90.000,E1 229.908} C_DIS
LIN {X -0.013,Y -151.972,Z 1031.252,A 0.000,B 0.000,C 90.000,E1 225.405} C_DIS
LIN {X 0.003,Y -150.215,Z 1031.237,A 0.000,B 0.000,C 90.000,E1 222.690} C_DIS
LIN {X -0.073,Y -146.980,Z 1031.212,A 0.000,B 0.000,C 90.000,E1 218.177} C_DIS
LIN {X 0.036,Y -145.566,Z 1031.197,A 0.000,B 0.000,C 90.000,E1 215.391} C_DIS
LIN {X 0.035,Y -142.957,Z 1031.171,A 0.000,B 0.000,C 90.000,E1 210.797} C_DIS
LIN {X -0.034,Y -141.583,Z 1031.151,A 0.000,B 0.000,C 90.000,E1 207.129} C_DIS
LIN {X 0.013,Y -139.417,Z 1031.115,A 0.000,B 0.000,C 90.000,E1 200.610} C_DIS
LIN {X 0.066,Y -139.142,Z 1031.104,A 0.000,B 0.000,C 90.000,E1 198.725} C_DIS
LIN {X -0.044,Y -138.347,Z 1031.057,A 0.000,B 0.000,C 90.000,E1 190.366} C_DIS
LIN {X -0.059,Y -139.491,Z 1031.006,A 0.000,B 0.000,C 90.000,E1 181.031} C_DIS
LIN {X 0.022,Y -141.099,Z 1030.975,A 0.000,B 0.000,C 90.000,E1 175.412} C_DIS
LIN {X -0.025,Y -142.479,Z 1030.959,A 0.000,B 0.000,C 90.000,E1 172.648} C_DIS
LIN {X 0.063,Y -144.727,Z 1030.933,A 0.000,B 0.000,C 90.000,E1 167.993} C_DIS
LIN {X 0.014,Y -147.330,Z 1030.913,A 0.000,B 0.000,C 90.000,E1 164.338} C_DIS
LIN {X 0.080,Y -150.653,Z 1030.888,A 0.000,B 0.000,C 90.000,E1 159.752} C_DIS
LIN {X -0.038,Y -154.131,Z 1030.868,A 0.000,B 0.000,C 90.000,E1 156.177} C_DIS
LIN {X 0.024,Y -157.558,Z 1030.848,A 0.000,B 0.000,C 90.000,E1 152.564} C_DIS
LIN {X 0.049,Y -161.799,Z 1030.828,A 0.000,B 0.000,C 90.000,E1 148.997} C_DIS
LIN {X 0.068,Y -165.992,Z 1030.808,A 0.000,B 0.000,C 90.000,E1 145.468} C_DIS
LIN {X 0.062,Y -170.988,Z 1030.789,A 0.000,B 0.000,C 90.000,E1 141.984} C_DIS
LIN {X -0.023,Y -175.859,Z 1030.770,A 0.000,B 0.000,C 90.000,E1 138.566} C_DIS
LIN {X -0.029,Y -181.463,Z 1030.751,A 0.000,B 0.000,C 90.000,E1 135.162} C_DIS
LIN {X 0.108,Y -186.974,Z 1030.732,A 0.000,B 0.000,C 90.000,E1 131.757} C_DIS
LIN {X 0.110,Y -190.089,Z 1030.723,A 0.000,B 0.000,C 90.000,E1 130.092} C_DIS
LIN {X -0.051,Y -197.293,Z 1030.700,A 0.000,B 0.000,C 90.000,E1 126.091} C_DIS
LIN {X -0.113,Y -302.837,Z 1030.700,A 0.000,B 0.000,C 90.000,E1 126.091} C_DIS
LIN {X -0.002,Y -305.462,Z 1030.700,A 0.000,B 0.000,C 90.000,E1 126.011} C_DIS
LIN {X -0.012,Y -308.661,Z 1030.699,A 0.000,B 0.000,C 90.000,E1 125.851} C_DIS
LIN {X 0.099,Y -312.223,Z 1030.697,A 0.000,B 0.000,C 90.000,E1 125.518} C_DIS
LIN {X 0.022,Y -315.832,Z 1030.695,A 0.000,B 0.000,C 90.000,E1 125.025} C_DIS
LIN {X 0.076,Y -317.455,Z 1030.693,A 0.000,B 0.000,C 90.000,E1 124.692} C_DIS
LIN {X -0.062,Y -319.782,Z 1030.689,A 0.000,B 0.000,C 90.000,E1 124.072} C_DIS
LIN {X 0.050,Y -331.026,Z 1030.672,A 0.000,B 0.000,C 90.000,E1 120.875} C_DIS
LIN {X -0.144,Y -342.547,Z 1030.656,A 0.000,B 0.000,C 90.000,E1 118.103} C_DIS
LIN {X -0.034,Y -355.498,Z 1030.641,A 0.000,B 0.000,C 90.000,E1 115.335} C_DIS
LIN {X -0.091,Y -368.306,Z 1030.627,A 0.000,B 0.000,C 90.000,E1 112.950} C_DIS
LIN {X -0.113,Y -382.425,Z 1030.614,A 0.000,B 0.000,C 90.000,E1 110.610} C_DIS
LIN {X -0.040,Y -397.955,Z 1030.602,A 0.000,B 0.000,C 90.000,E1 108.308} C_DIS
LIN {X -0.085,Y -415.009,Z 1030.589,A 0.000,B 0.000,C 90.000,E1 106.079} C_DIS
LIN {X 0.052,Y -433.707,Z 1030.577,A 0.000,B 0.000,C 90.000,E1 103.883} C_DIS
LIN {X -0.011,Y -453.653,Z 1030.566,A 0.000,B 0.000,C 90.000,E1 101.827} C_DIS
LIN {X 0.146,Y -466.427,Z 1030.559,A 0.000,B 0.000,C 90.000,E1 100.602} C_DIS
LIN {X 0.178,Y -468.696,Z 1030.558,A 0.000,B 0.000,C 90.000,E1 100.366} C_DIS
LIN {X 0.126,Y -470.408,Z 1030.556,A 0.000,B 0.000,C 90.000,E1 100.141} C_DIS
LIN {X -0.021,Y -471.832,Z 1030.555,A 0.000,B 0.000,C 90.000,E1 99.905} C_DIS
LIN {X -0.170,Y -472.893,Z 1030.554,A 0.000,B 0.000,C 90.000,E1 99.670} C_DIS
LIN {X -0.062,Y -474.131,Z 1030.551,A 0.000,B 0.000,C 90.000,E1 99.151} C_DIS
LIN {X 0.127,Y -474.364,Z 1030.548,A 0.000,B 0.000,C 90.000,E1 98.624} C_DIS
LIN {X -0.219,Y -473.630,Z 1030.545,A 0.000,B 0.000,C 90.000,E1 98.163} C_DIS
LIN {X -0.091,Y -471.815,Z 1030.542,A 0.000,B 0.000,C 90.000,E1 97.644} C_DIS
LIN {X 0.234,Y -470.397,Z 1030.541,A 0.000,B 0.000,C 90.000,E1 97.352} C_DIS
LIN {X -0.174,Y -458.074,Z 1030.531,A 0.000,B 0.000,C 90.000,E1 95.625} C_DIS
LIN {X 0.020,Y -442.018,Z 1030.518,A 0.000,B 0.000,C 90.000,E1 93.269} C_DIS
LIN {X 0.206,Y -427.192,Z 1030.505,A 0.000,B 0.000,C 90.000,E1 90.859} C_DIS
LIN {X 0.175,Y -410.765,Z 1030.488,A 0.000,B 0.000,C 90.000,E1 87.879} C_DIS
LIN {X -0.199,Y -401.905,Z 1030.479,A 0.000,B 0.000,C 90.000,E1 86.274} C_DIS
LIN {X 0.090,Y -392.929,Z 1030.470,A 0.000,B 0.000,C 90.000,E1 84.552} C_DIS
LIN {X -0.109,Y -382.080,Z 1030.459,A 0.000,B 0.000,C 90.000,E1 82.591} C_DIS
LIN {X -0.059,Y -374.157,Z 1030.451,A 0.000,B 0.000,C 90.000,E1 81.141} C_DIS
LIN {X -0.122,Y -365.944,Z 1030.443,A 0.000,B 0.000,C 90.000,E1 79.690} C_DIS
LIN {X 0.020,Y -354.329,Z 1030.431,A 0.000,B 0.000,C 90.000,E1 77.589} C_DIS
LIN {X -0.018,Y -341.174,Z 1030.418,A 0.000,B 0.000,C 90.000,E1 75.172} C_DIS
LIN {X 0.124,Y -328.394,Z 1030.404,A 0.000,B 0.000,C 90.000,E1 72.670} C_DIS
LIN {X 0.077,Y -314.470,Z 1030.388,A 0.000,B 0.000,C 90.000,E1 69.826} C_DIS
LIN {X 0.088,Y -302.542,Z 1030.374,A 0.000,B 0.000,C 90.000,E1 67.230} C_DIS
LIN {X -0.079,Y -293.810,Z 1030.363,A 0.000,B 0.000,C 90.000,E1 65.281} C_DIS
LIN {X 0.051,Y -282.373,Z 1030.348,A 0.000,B 0.000,C 90.000,E1 62.564} C_DIS
LIN {X -0.156,Y -272.593,Z 1030.334,A 0.000,B 0.000,C 90.000,E1 60.205} C_DIS
LIN {X -0.009,Y -261.551,Z 1030.319,A 0.000,B 0.000,C 90.000,E1 57.375} C_DIS
LIN {X 0.137,Y -250.845,Z 1030.303,A 0.000,B 0.000,C 90.000,E1 54.482} C_DIS
LIN {X -0.106,Y -239.479,Z 1030.285,A 0.000,B 0.000,C 90.000,E1 51.251} C_DIS
LIN {X -0.061,Y -228.790,Z 1030.266,A 0.000,B 0.000,C 90.000,E1 47.877} C_DIS
LIN {X -0.030,Y -218.858,Z 1030.247,A 0.000,B 0.000,C 90.000,E1 44.433} C_DIS
LIN {X 0.024,Y -210.403,Z 1030.229,A 0.000,B 0.000,C 90.000,E1 41.310} C_DIS
LIN {X -0.087,Y -202.533,Z 1030.212,A 0.000,B 0.000,C 90.000,E1 38.177} C_DIS
LIN {X -0.039,Y -195.209,Z 1030.194,A 0.000,B 0.000,C 90.000,E1 34.945} C_DIS
LIN {X -0.028,Y -188.569,Z 1030.176,A 0.000,B 0.000,C 90.000,E1 31.671} C_DIS
LIN {X -0.048,Y -182.677,Z 1030.157,A 0.000,B 0.000,C 90.000,E1 28.359} C_DIS
LIN {X 0.016,Y -177.592,Z 1030.139,A 0.000,B 0.000,C 90.000,E1 24.975} C_DIS
LIN {X -0.030,Y -173.316,Z 1030.120,A 0.000,B 0.000,C 90.000,E1 21.589} C_DIS
LIN {X 0.049,Y -169.724,Z 1030.101,A 0.000,B 0.000,C 90.000,E1 18.127} C_DIS
LIN {X -0.053,Y -166.278,Z 1030.077,A 0.000,B 0.000,C 90.000,E1 13.828} C_DIS
LIN {X -0.004,Y -163.507,Z 1030.048,A 0.000,B 0.000,C 90.000,E1 8.568} C_DIS
LIN {X 0.030,Y -164.338,Z 1029.953,A 0.000,B 0.000,C 90.000,E1 351.602} C_DIS
LIN {X 0.033,Y -167.596,Z 1029.924,A 0.000,B 0.000,C 90.000,E1 346.353} C_DIS
LIN {X 0.071,Y -171.374,Z 1029.900,A 0.000,B 0.000,C 90.000,E1 342.000} C_DIS
LIN {X -0.038,Y -175.191,Z 1029.881,A 0.000,B 0.000,C 90.000,E1 338.592} C_DIS
LIN {X -0.028,Y -179.829,Z 1029.862,A 0.000,B 0.000,C 90.000,E1 335.177} C_DIS
LIN {X 0.077,Y -185.291,Z 1029.843,A 0.000,B 0.000,C 90.000,E1 331.769} C_DIS
LIN {X 0.015,Y -191.608,Z 1029.825,A 0.000,B 0.000,C 90.000,E1 328.456} C_DIS
LIN {X -0.019,Y -198.663,Z 1029.807,A 0.000,B 0.000,C 90.000,E1 325.182} C_DIS
LIN {X -0.021,Y -206.275,Z 1029.789,A 0.000,B 0.000,C 90.000,E1 321.949} C_DIS
LIN {X -0.013,Y -214.471,Z 1029.771,A 0.000,B 0.000,C 90.000,E1 318.771} C_DIS
LIN {X 0.093,Y -224.438,Z 1029.751,A 0.000,B 0.000,C 90.000,E1 315.243} C_DIS
LIN {X 0.053,Y -234.332,Z 1029.734,A 0.000,B 0.000,C 90.000,E1 312.204} C_DIS
LIN {X 0.036,Y -241.291,Z 1029.724,A 0.000,B 0.000,C 90.000,E1 310.334} C_DIS
LIN {X 0.143,Y -250.719,Z 1029.712,A 0.000,B 0.000,C 90.000,E1 308.096} C_DIS
LIN {X 0.090,Y -259.645,Z 1029.702,A 0.000,B 0.000,C 90.000,E1 306.297} C_DIS
LIN {X -0.077,Y -275.559,Z 1029.686,A 0.000,B 0.000,C 90.000,E1 303.499} C_DIS
LIN {X 0.071,Y -294.907,Z 1029.669,A 0.000,B 0.000,C 90.000,E1 300.384} C_DIS
LIN {X -0.065,Y -315.969,Z 1029.652,A 0.000,B 0.000,C 90.000,E1 297.436} C_DIS
LIN {X -0.162,Y -328.804,Z 1029.643,A 0.000,B 0.000,C 90.000,E1 295.848} C_DIS
LIN {X 0.002,Y -347.492,Z 1029.632,A 0.000,B 0.000,C 90.000,E1 293.770} C_DIS
LIN {X -0.118,Y -369.392,Z 1029.620,A 0.000,B 0.000,C 90.000,E1 291.663} C_DIS
LIN {X -0.123,Y -385.998,Z 1029.612,A 0.000,B 0.000,C 90.000,E1 290.174} C_DIS
LIN {X 0.138,Y -402.450,Z 1029.604,A 0.000,B 0.000,C 90.000,E1 288.671} C_DIS
LIN {X 0.240,Y -413.055,Z 1029.599,A 0.000,B 0.000,C 90.000,E1 287.692} C_DIS
LIN {X 0.042,Y -420.710,Z 1029.594,A 0.000,B 0.000,C 90.000,E1 286.985} C_DIS
LIN {X 0.096,Y -428.250,Z 1029.590,A 0.000,B 0.000,C 90.000,E1 286.205} C_DIS
LIN {X 0.176,Y -437.990,Z 1029.584,A 0.000,B 0.000,C 90.000,E1 285.134} C_DIS
LIN {X -0.170,Y -447.097,Z 1029.578,A 0.000,B 0.000,C 90.000,E1 284.120} C_DIS
LIN {X 0.097,Y -453.463,Z 1029.574,A 0.000,B 0.000,C 90.000,E1 283.300} C_DIS
LIN {X -0.010,Y -459.363,Z 1029.570,A 0.000,B 0.000,C 90.000,E1 282.535} C_DIS
LIN {X -0.074,Y -464.690,Z 1029.565,A 0.000,B 0.000,C 90.000,E1 281.771} C_DIS
LIN {X -0.089,Y -469.496,Z 1029.561,A 0.000,B 0.000,C 90.000,E1 281.007} C_DIS
LIN {X -0.157,Y -473.712,Z 1029.557,A 0.000,B 0.000,C 90.000,E1 280.254} C_DIS
LIN {X -0.180,Y -477.311,Z 1029.553,A 0.000,B 0.000,C 90.000,E1 279.500} C_DIS
LIN {X -0.171,Y -480.366,Z 1029.548,A 0.000,B 0.000,C 90.000,E1 278.746} C_DIS
LIN {X 0.051,Y -482.090,Z 1029.546,A 0.000,B 0.000,C 90.000,E1 278.219} C_DIS
LIN {X 0.214,Y -483.568,Z 1029.543,A 0.000,B 0.000,C 90.000,E1 277.701} C_DIS
LIN {X -0.091,Y -484.798,Z 1029.540,A 0.000,B 0.000,C 90.000,E1 277.239} C_DIS
LIN {X 0.094,Y -485.834,Z 1029.537,A 0.000,B 0.000,C 90.000,E1 276.720} C_DIS
LIN {X -0.197,Y -486.647,Z 1029.535,A 0.000,B 0.000,C 90.000,E1 276.258} C_DIS
LIN {X 0.002,Y -487.169,Z 1029.532,A 0.000,B 0.000,C 90.000,E1 275.739} C_DIS
LIN {X 0.204,Y -487.337,Z 1029.529,A 0.000,B 0.000,C 90.000,E1 275.220} C_DIS
LIN {X -0.079,Y -487.068,Z 1029.526,A 0.000,B 0.000,C 90.000,E1 274.759} C_DIS
LIN {X 0.087,Y -486.308,Z 1029.524,A 0.000,B 0.000,C 90.000,E1 274.245} C_DIS
LIN {X -0.196,Y -485.035,Z 1029.521,A 0.000,B 0.000,C 90.000,E1 273.784} C_DIS
LIN {X -0.030,Y -483.149,Z 1029.518,A 0.000,B 0.000,C 90.000,E1 273.269} C_DIS
LIN {X 0.154,Y -480.614,Z 1029.515,A 0.000,B 0.000,C 90.000,E1 272.751} C_DIS
LIN {X -0.182,Y -477.321,Z 1029.513,A 0.000,B 0.000,C 90.000,E1 272.293} C_DIS
LIN {X -0.038,Y -473.118,Z 1029.510,A 0.000,B 0.000,C 90.000,E1 271.776} C_DIS
LIN {X 0.160,Y -468.237,Z 1029.507,A 0.000,B 0.000,C 90.000,E1 271.260} C_DIS
LIN {X -0.061,Y -462.452,Z 1029.504,A 0.000,B 0.000,C 90.000,E1 270.802} C_DIS
LIN {X 0.138,Y -456.263,Z 1029.502,A 0.000,B 0.000,C 90.000,E1 270.344} C_DIS
LIN {X -0.126,Y -449.559,Z 1029.500,A 0.000,B 0.000,C 90.000,E1 270.000} C_DIS
LIN {X 0.112,Y -442.240,Z 1029.498,A 0.000,B 0.000,C 90.000,E1 269.656} C_DIS
LIN {X -0.001,Y -434.477,Z 1029.497,A 0.000,B 0.000,C 90.000,E1 269.427} C_DIS
LIN {X -0.079,Y -425.560,Z 1029.496,A 0.000,B 0.000,C 90.000,E1 269.255} C_DIS
LIN {X -0.113,Y -416.925,Z 1029.495,A 0.000,B 0.000,C 90.000,E1 269.141} C_DIS
LIN {X 0.072,Y -406.569,Z 1029.495,A 0.000,B 0.000,C 90.000,E1 269.026} C_DIS
LIN {X 0.171,Y -398.217,Z 1029.494,A 0.000,B 0.000,C 90.000,E1 268.969} C_DIS
LIN {X 0.050,Y -181.315,Z 1029.494,A 0.000,B 0.000,C 90.000,E1 268.969} C_DIS
LIN {X 0.076,Y -180.901,Z 1029.474,A 0.000,B 0.000,C 90.000,E1 265.241} C_DIS
LIN {X 0.026,Y -180.228,Z 1029.464,A 0.000,B 0.000,C 90.000,E1 263.571} C_DIS
LIN {X -0.021,Y -179.041,Z 1029.446,A 0.000,B 0.000,C 90.000,E1 260.208} C_DIS
LIN {X 0.042,Y -178.711,Z 1029.441,A 0.000,B 0.000,C 90.000,E1 259.342} C_DIS
LIN {X -0.065,Y -175.759,Z 1029.413,A 0.000,B 0.000,C 90.000,E1 254.283} C_DIS
LIN {X -0.016,Y -171.943,Z 1029.384,A 0.000,B 0.000,C 90.000,E1 249.135} C_DIS
LIN {X -0.039,Y -171.327,Z 1029.379,A 0.000,B 0.000,C 90.000,E1 248.284} C_DIS
LIN {X 0.014,Y -167.584,Z 1029.355,A 0.000,B 0.000,C 90.000,E1 243.948} C_DIS
LIN {X -0.048,Y -166.218,Z 1029.346,A 0.000,B 0.000,C 90.000,E1 242.231} C_DIS
LIN {X -0.059,Y -162.981,Z 1029.326,A 0.000,B 0.000,C 90.000,E1 238.742} C_DIS
LIN {X -0.012,Y -160.896,Z 1029.312,A 0.000,B 0.000,C 90.000,E1 236.087} C_DIS
LIN {X -0.033,Y -157.664,Z 1029.292,A 0.000,B 0.000,C 90.000,E1 232.557} C_DIS
LIN {X -0.095,Y -155.703,Z 1029.277,A 0.000,B 0.000,C 90.000,E1 229.908} C_DIS
LIN {X -0.039,Y -151.965,Z 1029.252,A 0.000,B 0.000,C 90.000,E1 225.405} C_DIS
LIN {X -0.023,Y -150.207,Z 1029.237,A 0.000,B 0.000,C 90.000,E1 222.690} C_DIS
LIN {X -0.008,Y -146.974,Z 1029.212,A 0.000,B 0.000,C 90.000,E1 218.141} C_DIS
LIN {X 0.011,Y -145.560,Z 1029.197,A 0.000,B 0.000,C 90.000,E1 215.391} C_DIS
LIN {X 0.009,Y -142.953,Z 1029.171,A 0.000,B 0.000,C 90.000,E1 210.797} C_DIS
LIN {X -0.059,Y -141.578,Z 1029.151,A 0.000,B 0.000,C 90.000,E1 207.129} C_DIS
LIN {X -0.012,Y -139.415,Z 1029.115,A 0.000,B 0.000,C 90.000,E1 200.610} C_DIS
LIN {X 0.040,Y -139.139,Z 1029.104,A 0.000,B 0.000,C 90.000,E1 198.725} C_DIS
LIN {X 0.067,Y -138.348,Z 1029.057,A 0.000,B 0.000,C 90.000,E1 190.310} C_DIS
LIN {X 0.055,Y -139.492,Z 1029.005,A 0.000,B 0.000,C 90.000,E1 180.974} C_DIS
LIN {X -0.004,Y -141.104,Z 1028.974,A 0.000,B 0.000,C 90.000,E1 175.412} C_DIS
LIN {X -0.051,Y -142.483,Z 1028.959,A 0.000,B 0.000,C 90.000,E1 172.648} C_DIS
LIN {X 0.038,Y -144.733,Z 1028.933,A 0.000,B 0.000,C 90.000,E1 167.993} C_DIS
LIN {X -0.011,Y -147.337,Z 1028.913,A 0.000,B 0.000,C 90.000,E1 164.338} C_DIS
LIN {X 0.054,Y -150.661,Z 1028.888,A 0.000,B 0.000,C 90.000,E1 159.752} C_DIS
LIN {X -0.065,Y -154.139,Z 1028.868,A 0.000,B 0.000,C 90.000,E1 156.177} C_DIS
LIN {X -0.003,Y -157.568,Z 1028.848,A 0.000,B 0.000,C 90.000,E1 152.564} C_DIS
LIN {X 0.022,Y -161.812,Z 1028.828,A 0.000,B 0.000,C 90.000,E1 148.997} C_DIS
LIN {X 0.041,Y -166.004,Z 1028.808,A 0.000,B 0.000,C 90.000,E1 145.468} C_DIS
LIN {X 0.034,Y -171.003,Z 1028.789,A 0.000,B 0.000,C 90.000,E1 141.984} C_DIS
LIN {X -0.051,Y -175.873,Z 1028.770,A 0.000,B 0.000,C 90.000,E1 138.566} C_DIS
LIN {X -0.059,Y -181.477,Z 1028.751,A 0.000,B 0.000,C 90.000,E1 135.162} C_DIS
LIN {X 0.078,Y -186.991,Z 1028.732,A 0.000,B 0.000,C 90.000,E1 131.757} C_DIS
LIN {X 0.080,Y -190.107,Z 1028.723,A 0.000,B 0.000,C 90.000,E1 130.092} C_DIS
LIN {X 0.090,Y -197.213,Z 1028.701,A 0.000,B 0.000,C 90.000,E1 126.091} C_DIS
LIN {X 0.104,Y -302.385,Z 1028.701,A 0.000,B 0.000,C 90.000,E1 126.091} C_DIS
LIN {X -0.049,Y -306.500,Z 1028.700,A 0.000,B 0.000,C 90.000,E1 126.011} C_DIS
LIN {X 0.144,Y -309.314,Z 1028.699,A 0.000,B 0.000,C 90.000,E1 125.804} C_DIS
LIN {X 0.132,Y -313.043,Z 1028.697,A 0.000,B 0.000,C 90.000,E1 125.438} C_DIS
LIN {X 0.036,Y -316.556,Z 1028.694,A 0.000,B 0.000,C 90.000,E1 124.898} C_DIS
LIN {X -0.169,Y -317.989,Z 1028.692,A 0.000,B 0.000,C 90.000,E1 124.612} C_DIS
LIN {X 0.091,Y -331.467,Z 1028.671,A 0.000,B 0.000,C 90.000,E1 120.747} C_DIS
LIN {X -0.087,Y -343.048,Z 1028.655,A 0.000,B 0.000,C 90.000,E1 117.975} C_DIS
LIN {X 0.040,Y -356.063,Z 1028.640,A 0.000,B 0.000,C 90.000,E1 115.207} C_DIS
LIN {X -0.001,Y -368.931,Z 1028.627,A 0.000,B 0.000,C 90.000,E1 112.823} C_DIS
LIN {X -0.007,Y -383.115,Z 1028.614,A 0.000,B 0.000,C 90.000,E1 110.482} C_DIS
LIN {X 0.084,Y -398.716,Z 1028.601,A 0.000,B 0.000,C 90.000,E1 108.181} C_DIS
LIN {X -0.059,Y -415.845,Z 1028.589,A 0.000,B 0.000,C 90.000,E1 105.969} C_DIS
LIN {X 0.111,Y -434.625,Z 1028.577,A 0.000,B 0.000,C 90.000,E1 103.772} C_DIS
LIN {X 0.118,Y -454.607,Z 1028.565,A 0.000,B 0.000,C 90.000,E1 101.715} C_DIS
LIN {X -0.135,Y -467.369,Z 1028.558,A 0.000,B 0.000,C 90.000,E1 100.546} C_DIS
LIN {X -0.139,Y -469.431,Z 1028.557,A 0.000,B 0.000,C 90.000,E1 100.310} C_DIS
LIN {X -0.143,Y -470.995,Z 1028.556,A 0.000,B 0.000,C 90.000,E1 100.074} C_DIS
LIN {X 0.094,Y -472.269,Z 1028.554,A 0.000,B 0.000,C 90.000,E1 99.792} C_DIS
LIN {X -0.052,Y -473.207,Z 1028.553,A 0.000,B 0.000,C 90.000,E1 99.557} C_DIS
LIN {X 0.134,Y -474.244,Z 1028.550,A 0.000,B 0.000,C 90.000,E1 99.029} C_DIS
LIN {X -0.218,Y -474.293,Z 1028.547,A 0.000,B 0.000,C 90.000,E1 98.568} C_DIS
LIN {X -0.092,Y -473.368,Z 1028.545,A 0.000,B 0.000,C 90.000,E1 98.049} C_DIS
LIN {X 0.036,Y -471.315,Z 1028.542,A 0.000,B 0.000,C 90.000,E1 97.530} C_DIS
LIN {X 0.157,Y -467.958,Z 1028.539,A 0.000,B 0.000,C 90.000,E1 97.011} C_DIS
LIN {X -0.059,Y -457.420,Z 1028.531,A 0.000,B 0.000,C 90.000,E1 95.511} C_DIS
LIN {X -0.209,Y -436.275,Z 1028.513,A 0.000,B 0.000,C 90.000,E1 92.407} C_DIS
LIN {X -0.059,Y -420.459,Z 1028.498,A 0.000,B 0.000,C 90.000,E1 89.714} C_DIS
LIN {X -0.095,Y -408.775,Z 1028.486,A 0.000,B 0.000,C 90.000,E1 87.535} C_DIS
LIN {X -0.032,Y -398.382,Z 1028.475,A 0.000,B 0.000,C 90.000,E1 85.584} C_DIS
LIN {X -0.161,Y -389.265,Z 1028.466,A 0.000,B 0.000,C 90.000,E1 83.913} C_DIS
LIN {X -0.042,Y -378.380,Z 1028.455,A 0.000,B 0.000,C 90.000,E1 81.894} C_DIS
LIN {X -0.047,Y -368.654,Z 1028.445,A 0.000,B 0.000,C 90.000,E1 80.151} C_DIS
LIN {X 0.157,Y -357.002,Z 1028.434,A 0.000,B 0.000,C 90.000,E1 78.049} C_DIS
LIN {X -0.151,Y -345.437,Z 1028.422,A 0.000,B 0.000,C 90.000,E1 75.992} C_DIS
LIN {X 0.018,Y -332.571,Z 1028.408,A 0.000,B 0.000,C 90.000,E1 73.504} C_DIS
LIN {X -0.015,Y -318.485,Z 1028.393,A 0.000,B 0.000,C 90.000,E1 70.678} C_DIS
LIN {X -0.017,Y -306.408,Z 1028.378,A 0.000,B 0.000,C 90.000,E1 68.103} C_DIS
LIN {X 0.043,Y -296.189,Z 1028.366,A 0.000,B 0.000,C 90.000,E1 65.793} C_DIS
LIN {X -0.027,Y -284.662,Z 1028.351,A 0.000,B 0.000,C 90.000,E1 63.127} C_DIS
LIN {X 0.062,Y -274.847,Z 1028.337,A 0.000,B 0.000,C 90.000,E1 60.717} C_DIS
LIN {X -0.016,Y -263.753,Z 1028.322,A 0.000,B 0.000,C 90.000,E1 57.946} C_DIS
LIN {X -0.029,Y -252.965,Z 1028.306,A 0.000,B 0.000,C 90.000,E1 55.102} C_DIS
LIN {X -0.012,Y -241.457,Z 1028.288,A 0.000,B 0.000,C 90.000,E1 51.823} C_DIS
LIN {X -0.063,Y -230.637,Z 1028.269,A 0.000,B 0.000,C 90.000,E1 48.485} C_DIS
LIN {X 0.022,Y -220.547,Z 1028.250,A 0.000,B 0.000,C 90.000,E1 45.040} C_DIS
LIN {X 0.104,Y -212.003,Z 1028.233,A 0.000,B 0.000,C 90.000,E1 41.919} C_DIS
LIN {X -0.129,Y -203.973,Z 1028.216,A 0.000,B 0.000,C 90.000,E1 38.830} C_DIS
LIN {X -0.043,Y -196.543,Z 1028.198,A 0.000,B 0.000,C 90.000,E1 35.598} C_DIS
LIN {X -0.051,Y -189.737,Z 1028.180,A 0.000,B 0.000,C 90.000,E1 32.339} C_DIS
LIN {X 0.046,Y -183.694,Z 1028.161,A 0.000,B 0.000,C 90.000,E1 28.999} C_DIS
LIN {X -0.032,Y -178.444,Z 1028.143,A 0.000,B 0.000,C 90.000,E1 25.668} C_DIS
LIN {X -0.055,Y -174.034,Z 1028.124,A 0.000,B 0.000,C 90.000,E1 22.280} C_DIS
LIN {X -0.058,Y -170.306,Z 1028.105,A 0.000,B 0.000,C 90.000,E1 18.852} C_DIS
LIN {X 0.069,Y -166.658,Z 1028.081,A 0.000,B 0.000,C 90.000,E1 14.481} C_DIS
LIN {X 0.002,Y -163.707,Z 1028.052,A 0.000,B 0.000,C 90.000,E1 9.265} C_DIS
LIN {X 0.000,Y -162.079,Z 1028.000,A 0.000,B 0.000,C 90.000,E1 360.000} C_DIS
LIN {X 0.057,Y -163.899,Z 1027.958,A 0.000,B 0.000,C 90.000,E1 352.470} C_DIS
LIN {X 0.017,Y -166.907,Z 1027.929,A 0.000,B 0.000,C 90.000,E1 347.229} C_DIS
LIN {X -0.057,Y -170.475,Z 1027.905,A 0.000,B 0.000,C 90.000,E1 342.906} C_DIS
LIN {X -0.026,Y -174.112,Z 1027.886,A 0.000,B 0.000,C 90.000,E1 339.444} C_DIS
LIN {X 0.055,Y -178.535,Z 1027.867,A 0.000,B 0.000,C 90.000,E1 335.997} C_DIS
LIN {X 0.045,Y -183.818,Z 1027.848,A 0.000,B 0.000,C 90.000,E1 332.615} C_DIS
LIN {X 0.012,Y -189.946,Z 1027.829,A 0.000,B 0.000,C 90.000,E1 329.282} C_DIS
LIN {X -0.067,Y -196.798,Z 1027.811,A 0.000,B 0.000,C 90.000,E1 326.008} C_DIS
LIN {X -0.075,Y -204.293,Z 1027.793,A 0.000,B 0.000,C 90.000,E1 322.763} C_DIS
LIN {X 0.035,Y -212.311,Z 1027.775,A 0.000,B 0.000,C 90.000,E1 319.542} C_DIS
LIN {X -0.075,Y -222.100,Z 1027.756,A 0.000,B 0.000,C 90.000,E1 316.053} C_DIS
LIN {X -0.024,Y -231.690,Z 1027.739,A 0.000,B 0.000,C 90.000,E1 312.975} C_DIS
LIN {X 0.069,Y -238.359,Z 1027.728,A 0.000,B 0.000,C 90.000,E1 311.067} C_DIS
LIN {X 0.126,Y -245.825,Z 1027.718,A 0.000,B 0.000,C 90.000,E1 309.197} C_DIS
LIN {X 0.131,Y -252.388,Z 1027.710,A 0.000,B 0.000,C 90.000,E1 307.729} C_DIS
LIN {X 0.097,Y -261.527,Z 1027.700,A 0.000,B 0.000,C 90.000,E1 305.931} C_DIS
LIN {X -0.179,Y -277.614,Z 1027.684,A 0.000,B 0.000,C 90.000,E1 303.166} C_DIS
LIN {X 0.034,Y -297.194,Z 1027.667,A 0.000,B 0.000,C 90.000,E1 300.050} C_DIS
LIN {X 0.091,Y -318.544,Z 1027.651,A 0.000,B 0.000,C 90.000,E1 297.078} C_DIS
LIN {X -0.150,Y -331.528,Z 1027.642,A 0.000,B 0.000,C 90.000,E1 295.540} C_DIS
LIN {X -0.095,Y -347.803,Z 1027.632,A 0.000,B 0.000,C 90.000,E1 293.770} C_DIS
LIN {X 0.199,Y -369.801,Z 1027.620,A 0.000,B 0.000,C 90.000,E1 291.589} C_DIS
LIN {X 0.073,Y -386.388,Z 1027.612,A 0.000,B 0.000,C 90.000,E1 290.120} C_DIS
LIN {X -0.044,Y -402.816,Z 1027.604,A 0.000,B 0.000,C 90.000,E1 288.671} C_DIS
LIN {X 0.021,Y -413.425,Z 1027.598,A 0.000,B 0.000,C 90.000,E1 287.692} C_DIS
LIN {X -0.097,Y -421.072,Z 1027.594,A 0.000,B 0.000,C 90.000,E1 286.968} C_DIS
LIN {X -0.201,Y -428.605,Z 1027.590,A 0.000,B 0.000,C 90.000,E1 286.205} C_DIS
LIN {X -0.140,Y -438.302,Z 1027.584,A 0.000,B 0.000,C 90.000,E1 285.134} C_DIS
LIN {X -0.055,Y -447.368,Z 1027.578,A 0.000,B 0.000,C 90.000,E1 284.064} C_DIS
LIN {X -0.224,Y -453.727,Z 1027.574,A 0.000,B 0.000,C 90.000,E1 283.300} C_DIS
LIN {X 0.116,Y -459.582,Z 1027.569,A 0.000,B 0.000,C 90.000,E1 282.479} C_DIS
LIN {X 0.058,Y -464.906,Z 1027.565,A 0.000,B 0.000,C 90.000,E1 281.715} C_DIS
LIN {X 0.047,Y -469.706,Z 1027.561,A 0.000,B 0.000,C 90.000,E1 280.950} C_DIS
LIN {X -0.017,Y -473.923,Z 1027.557,A 0.000,B 0.000,C 90.000,E1 280.197} C_DIS
LIN {X -0.036,Y -477.511,Z 1027.552,A 0.000,B 0.000,C 90.000,E1 279.443} C_DIS
LIN {X 0.048,Y -480.547,Z 1027.548,A 0.000,B 0.000,C 90.000,E1 278.681} C_DIS
LIN {X 0.200,Y -482.267,Z 1027.546,A 0.000,B 0.000,C 90.000,E1 278.163} C_DIS
LIN {X -0.114,Y -483.729,Z 1027.543,A 0.000,B 0.000,C 90.000,E1 277.701} C_DIS
LIN {X 0.063,Y -484.962,Z 1027.540,A 0.000,B 0.000,C 90.000,E1 277.182} C_DIS
LIN {X -0.234,Y -485.980,Z 1027.537,A 0.000,B 0.000,C 90.000,E1 276.720} C_DIS
LIN {X -0.041,Y -486.792,Z 1027.534,A 0.000,B 0.000,C 90.000,E1 276.201} C_DIS
LIN {X 0.160,Y -487.321,Z 1027.532,A 0.000,B 0.000,C 90.000,E1 275.682} C_DIS
LIN {X -0.123,Y -487.492,Z 1027.529,A 0.000,B 0.000,C 90.000,E1 275.220} C_DIS
LIN {X 0.082,Y -487.169,Z 1027.526,A 0.000,B 0.000,C 90.000,E1 274.702} C_DIS
LIN {X -0.237,Y -486.402,Z 1027.523,A 0.000,B 0.000,C 90.000,E1 274.245} C_DIS
LIN {X -0.033,Y -485.123,Z 1027.521,A 0.000,B 0.000,C 90.000,E1 273.726} C_DIS
LIN {X 0.132,Y -483.212,Z 1027.518,A 0.000,B 0.000,C 90.000,E1 273.212} C_DIS
LIN {X -0.164,Y -480.615,Z 1027.515,A 0.000,B 0.000,C 90.000,E1 272.751} C_DIS
LIN {X -0.020,Y -477.275,Z 1027.512,A 0.000,B 0.000,C 90.000,E1 272.236} C_DIS
LIN {X 0.122,Y -473.117,Z 1027.510,A 0.000,B 0.000,C 90.000,E1 271.718} C_DIS
LIN {X 0.224,Y -468.026,Z 1027.507,A 0.000,B 0.000,C 90.000,E1 271.203} C_DIS
LIN {X 0.034,Y -462.215,Z 1027.504,A 0.000,B 0.000,C 90.000,E1 270.745} C_DIS
LIN {X 0.144,Y -459.281,Z 1027.503,A 0.000,B 0.000,C 90.000,E1 270.516} C_DIS
LIN {X 0.154,Y -452.861,Z 1027.501,A 0.000,B 0.000,C 90.000,E1 270.115} C_DIS
LIN {X 0.199,Y -445.979,Z 1027.499,A 0.000,B 0.000,C 90.000,E1 269.771} C_DIS
LIN {X -0.133,Y -438.389,Z 1027.497,A 0.000,B 0.000,C 90.000,E1 269.542} C_DIS
LIN {X 0.031,Y -430.328,Z 1027.496,A 0.000,B 0.000,C 90.000,E1 269.312} C_DIS
LIN {X 0.204,Y -421.631,Z 1027.495,A 0.000,B 0.000,C 90.000,E1 269.141} C_DIS
LIN {X -0.131,Y -412.174,Z 1027.495,A 0.000,B 0.000,C 90.000,E1 269.083} C_DIS
LIN {X 0.065,Y -397.883,Z 1027.494,A 0.000,B 0.000,C 90.000,E1 268.969} C_DIS
LIN {X 0.002,Y -181.311,Z 1027.494,A 0.000,B 0.000,C 90.000,E1 268.969} C_DIS
LIN {X 0.029,Y -180.900,Z 1027.474,A 0.000,B 0.000,C 90.000,E1 265.241} C_DIS
LIN {X -0.021,Y -180.222,Z 1027.464,A 0.000,B 0.000,C 90.000,E1 263.571} C_DIS
LIN {X -0.068,Y -179.038,Z 1027.445,A 0.000,B 0.000,C 90.000,E1 260.208} C_DIS
LIN {X -0.005,Y -178.701,Z 1027.441,A 0.000,B 0.000,C 90.000,E1 259.342} C_DIS
LIN {X 0.105,Y -175.750,Z 1027.412,A 0.000,B 0.000,C 90.000,E1 254.212} C_DIS
LIN {X -0.061,Y -171.933,Z 1027.384,A 0.000,B 0.000,C 90.000,E1 249.135} C_DIS
LIN {X -0.085,Y -171.313,Z 1027.379,A 0.000,B 0.000,C 90.000,E1 248.284} C_DIS
LIN {X -0.032,Y -167.572,Z 1027.355,A 0.000,B 0.000,C 90.000,E1 243.948} C_DIS
LIN {X -0.092,Y -166.202,Z 1027.346,A 0.000,B 0.000,C 90.000,E1 242.231} C_DIS
LIN {X -0.103,Y -162.969,Z 1027.326,A 0.000,B 0.000,C 90.000,E1 238.742} C_DIS
LIN {X -0.055,Y -160.880,Z 1027.312,A 0.000,B 0.000,C 90.000,E1 236.087} C_DIS
LIN {X -0.077,Y -157.651,Z 1027.292,A 0.000,B 0.000,C 90.000,E1 232.557} C_DIS
LIN {X 0.082,Y -155.689,Z 1027.277,A 0.000,B 0.000,C 90.000,E1 229.828} C_DIS
LIN {X -0.083,Y -151.954,Z 1027.252,A 0.000,B 0.000,C 90.000,E1 225.405} C_DIS
LIN {X -0.065,Y -150.194,Z 1027.237,A 0.000,B 0.000,C 90.000,E1 222.690} C_DIS
LIN {X 0.066,Y -146.964,Z 1027.212,A 0.000,B 0.000,C 90.000,E1 218.096} C_DIS
LIN {X -0.031,Y -145.552,Z 1027.197,A 0.000,B 0.000,C 90.000,E1 215.391} C_DIS
LIN {X -0.031,Y -142.945,Z 1027.171,A 0.000,B 0.000,C 90.000,E1 210.797} C_DIS
LIN {X 0.026,Y -141.570,Z 1027.151,A 0.000,B 0.000,C 90.000,E1 207.078} C_DIS
LIN {X -0.052,Y -139.412,Z 1027.114,A 0.000,B 0.000,C 90.000,E1 200.610} C_DIS
LIN {X 0.000,Y -139.135,Z 1027.104,A 0.000,B 0.000,C 90.000,E1 198.725} C_DIS
LIN {X 0.027,Y -138.350,Z 1027.057,A 0.000,B 0.000,C 90.000,E1 190.310} C_DIS
LIN {X 0.015,Y -139.494,Z 1027.005,A 0.000,B 0.000,C 90.000,E1 180.974} C_DIS
LIN {X -0.045,Y -141.112,Z 1026.974,A 0.000,B 0.000,C 90.000,E1 175.412} C_DIS
LIN {X 0.050,Y -142.490,Z 1026.959,A 0.000,B 0.000,C 90.000,E1 172.591} C_DIS
LIN {X -0.003,Y -144.743,Z 1026.933,A 0.000,B 0.000,C 90.000,E1 167.993} C_DIS
LIN {X -0.053,Y -147.350,Z 1026.913,A 0.000,B 0.000,C 90.000,E1 164.338} C_DIS
LIN {X 0.012,Y -150.675,Z 1026.888,A 0.000,B 0.000,C 90.000,E1 159.752} C_DIS
LIN {X 0.032,Y -154.154,Z 1026.867,A 0.000,B 0.000,C 90.000,E1 156.125} C_DIS
LIN {X 0.026,Y -157.586,Z 1026.848,A 0.000,B 0.000,C 90.000,E1 152.538} C_DIS
LIN {X -0.023,Y -161.833,Z 1026.828,A 0.000,B 0.000,C 90.000,E1 148.997} C_DIS
LIN {X -0.005,Y -166.025,Z 1026.808,A 0.000,B 0.000,C 90.000,E1 145.468} C_DIS
LIN {X -0.013,Y -171.026,Z 1026.789,A 0.000,B 0.000,C 90.000,E1 141.984} C_DIS
LIN {X 0.018,Y -175.896,Z 1026.770,A 0.000,B 0.000,C 90.000,E1 138.528} C_DIS
LIN {X 0.023,Y -181.500,Z 1026.751,A 0.000,B 0.000,C 90.000,E1 135.121} C_DIS
LIN {X 0.030,Y -187.017,Z 1026.732,A 0.000,B 0.000,C 90.000,E1 131.757} C_DIS
LIN {X 0.031,Y -190.136,Z 1026.723,A 0.000,B 0.000,C 90.000,E1 130.092} C_DIS
LIN {X -0.042,Y -197.133,Z 1026.701,A 0.000,B 0.000,C 90.000,E1 126.171} C_DIS
LIN {X -0.099,Y -302.224,Z 1026.701,A 0.000,B 0.000,C 90.000,E1 126.171} C_DIS
LIN {X -0.128,Y -307.418,Z 1026.700,A 0.000,B 0.000,C 90.000,E1 126.011} C_DIS
LIN {X -0.099,Y -310.202,Z 1026.699,A 0.000,B 0.000,C 90.000,E1 125.804} C_DIS
LIN {X -0.012,Y -313.980,Z 1026.696,A 0.000,B 0.000,C 90.000,E1 125.358} C_DIS
LIN {X 0.118,Y -315.876,Z 1026.695,A 0.000,B 0.000,C 90.000,E1 125.025} C_DIS
LIN {X -0.011,Y -317.365,Z 1026.693,A 0.000,B 0.000,C 90.000,E1 124.739} C_DIS
LIN {X -0.144,Y -319.634,Z 1026.689,A 0.000,B 0.000,C 90.000,E1 124.119} C_DIS
LIN {X -0.048,Y -330.860,Z 1026.672,A 0.000,B 0.000,C 90.000,E1 120.924} C_DIS
LIN {X 0.046,Y -342.363,Z 1026.656,A 0.000,B 0.000,C 90.000,E1 118.103} C_DIS
LIN {X 0.154,Y -355.300,Z 1026.641,A 0.000,B 0.000,C 90.000,E1 115.335} C_DIS
LIN {X 0.098,Y -368.091,Z 1026.628,A 0.000,B 0.000,C 90.000,E1 112.950} C_DIS
LIN {X 0.078,Y -382.194,Z 1026.615,A 0.000,B 0.000,C 90.000,E1 110.610} C_DIS
LIN {X 0.152,Y -397.705,Z 1026.602,A 0.000,B 0.000,C 90.000,E1 108.308} C_DIS
LIN {X 0.108,Y -414.739,Z 1026.589,A 0.000,B 0.000,C 90.000,E1 106.079} C_DIS
LIN {X -0.173,Y -433.415,Z 1026.577,A 0.000,B 0.000,C 90.000,E1 103.939} C_DIS
LIN {X 0.166,Y -453.365,Z 1026.566,A 0.000,B 0.000,C 90.000,E1 101.827} C_DIS
LIN {X -0.119,Y -466.109,Z 1026.559,A 0.000,B 0.000,C 90.000,E1 100.658} C_DIS
LIN {X -0.112,Y -468.470,Z 1026.558,A 0.000,B 0.000,C 90.000,E1 100.423} C_DIS
LIN {X 0.174,Y -470.332,Z 1026.556,A 0.000,B 0.000,C 90.000,E1 100.141} C_DIS
LIN {X 0.081,Y -471.742,Z 1026.555,A 0.000,B 0.000,C 90.000,E1 99.905} C_DIS
LIN {X 0.259,Y -473.596,Z 1026.552,A 0.000,B 0.000,C 90.000,E1 99.378} C_DIS
LIN {X -0.102,Y -474.353,Z 1026.549,A 0.000,B 0.000,C 90.000,E1 98.916} C_DIS
LIN {X 0.020,Y -474.138,Z 1026.547,A 0.000,B 0.000,C 90.000,E1 98.398} C_DIS
LIN {X 0.211,Y -472.927,Z 1026.544,A 0.000,B 0.000,C 90.000,E1 97.871} C_DIS
LIN {X 0.007,Y -471.891,Z 1026.542,A 0.000,B 0.000,C 90.000,E1 97.644} C_DIS
LIN {X -0.132,Y -470.500,Z 1026.541,A 0.000,B 0.000,C 90.000,E1 97.409} C_DIS
LIN {X -0.080,Y -458.218,Z 1026.531,A 0.000,B 0.000,C 90.000,E1 95.625} C_DIS
LIN {X 0.119,Y -442.142,Z 1026.518,A 0.000,B 0.000,C 90.000,E1 93.269} C_DIS
LIN {X -0.127,Y -427.280,Z 1026.505,A 0.000,B 0.000,C 90.000,E1 90.917} C_DIS
LIN {X -0.136,Y -410.901,Z 1026.488,A 0.000,B 0.000,C 90.000,E1 87.936} C_DIS
LIN {X -0.100,Y -402.039,Z 1026.479,A 0.000,B 0.000,C 90.000,E1 86.274} C_DIS
LIN {X -0.202,Y -393.038,Z 1026.470,A 0.000,B 0.000,C 90.000,E1 84.609} C_DIS
LIN {X -0.015,Y -382.194,Z 1026.459,A 0.000,B 0.000,C 90.000,E1 82.591} C_DIS
LIN {X 0.039,Y -374.268,Z 1026.451,A 0.000,B 0.000,C 90.000,E1 81.141} C_DIS
LIN {X -0.041,Y -364.415,Z 1026.441,A 0.000,B 0.000,C 90.000,E1 79.398} C_DIS
LIN {X 0.064,Y -352.761,Z 1026.429,A 0.000,B 0.000,C 90.000,E1 77.297} C_DIS
LIN {X 0.072,Y -339.654,Z 1026.416,A 0.000,B 0.000,C 90.000,E1 74.866} C_DIS
LIN {X -0.095,Y -328.522,Z 1026.404,A 0.000,B 0.000,C 90.000,E1 72.725} C_DIS
LIN {X -0.129,Y -314.646,Z 1026.388,A 0.000,B 0.000,C 90.000,E1 69.880} C_DIS
LIN {X 0.076,Y -301.209,Z 1026.372,A 0.000,B 0.000,C 90.000,E1 66.922} C_DIS
LIN {X 0.138,Y -291.022,Z 1026.359,A 0.000,B 0.000,C 90.000,E1 64.588} C_DIS
LIN {X 0.067,Y -279.650,Z 1026.344,A 0.000,B 0.000,C 90.000,E1 61.897} C_DIS
LIN {X 0.044,Y -269.884,Z 1026.331,A 0.000,B 0.000,C 90.000,E1 59.488} C_DIS
LIN {X -0.107,Y -258.902,Z 1026.315,A 0.000,B 0.000,C 90.000,E1 56.707} C_DIS
LIN {X -0.087,Y -248.280,Z 1026.299,A 0.000,B 0.000,C 90.000,E1 53.829} C_DIS
LIN {X -0.056,Y -237.069,Z 1026.281,A 0.000,B 0.000,C 90.000,E1 50.517} C_DIS
LIN {X -0.094,Y -226.557,Z 1026.262,A 0.000,B 0.000,C 90.000,E1 47.148} C_DIS
LIN {X 0.124,Y -217.741,Z 1026.245,A 0.000,B 0.000,C 90.000,E1 44.028} C_DIS
LIN {X 0.005,Y -209.302,Z 1026.227,A 0.000,B 0.000,C 90.000,E1 40.943} C_DIS
LIN {X -0.130,Y -201.438,Z 1026.210,A 0.000,B 0.000,C 90.000,E1 37.810} C_DIS
LIN {X 0.048,Y -194.185,Z 1026.192,A 0.000,B 0.000,C 90.000,E1 34.532} C_DIS
LIN {X 0.032,Y -187.598,Z 1026.174,A 0.000,B 0.000,C 90.000,E1 31.258} C_DIS
LIN {X -0.104,Y -181.826,Z 1026.155,A 0.000,B 0.000,C 90.000,E1 27.975} C_DIS
LIN {X -0.057,Y -176.849,Z 1026.136,A 0.000,B 0.000,C 90.000,E1 24.591} C_DIS
LIN {X 0.036,Y -172.705,Z 1026.118,A 0.000,B 0.000,C 90.000,E1 21.153} C_DIS
LIN {X 0.094,Y -169.185,Z 1026.099,A 0.000,B 0.000,C 90.000,E1 17.692} C_DIS
LIN {X -0.074,Y -165.836,Z 1026.074,A 0.000,B 0.000,C 90.000,E1 13.411} C_DIS
LIN {X -0.073,Y -163.221,Z 1026.045,A 0.000,B 0.000,C 90.000,E1 8.163} C_DIS
LIN {X 0.054,Y -163.841,Z 1025.958,A 0.000,B 0.000,C 90.000,E1 352.470} C_DIS
LIN {X 0.012,Y -166.841,Z 1025.929,A 0.000,B 0.000,C 90.000,E1 347.229} C_DIS
LIN {X -0.064,Y -170.415,Z 1025.905,A 0.000,B 0.000,C 90.000,E1 342.906} C_DIS
LIN {X -0.035,Y -174.058,Z 1025.886,A 0.000,B 0.000,C 90.000,E1 339.444} C_DIS
LIN {X 0.044,Y -178.502,Z 1025.867,A 0.000,B 0.000,C 90.000,E1 335.997} C_DIS
LIN {X 0.034,Y -183.803,Z 1025.848,A 0.000,B 0.000,C 90.000,E1 332.615} C_DIS
LIN {X 0.000,Y -189.939,Z 1025.829,A 0.000,B 0.000,C 90.000,E1 329.282} C_DIS
LIN {X -0.080,Y -196.786,Z 1025.811,A 0.000,B 0.000,C 90.000,E1 326.008} C_DIS
LIN {X -0.051,Y -205.254,Z 1025.791,A 0.000,B 0.000,C 90.000,E1 322.351} C_DIS
LIN {X 0.065,Y -213.330,Z 1025.773,A 0.000,B 0.000,C 90.000,E1 319.138} C_DIS
LIN {X -0.014,Y -223.198,Z 1025.754,A 0.000,B 0.000,C 90.000,E1 315.648} C_DIS
LIN {X -0.090,Y -232.919,Z 1025.737,A 0.000,B 0.000,C 90.000,E1 312.609} C_DIS
LIN {X 0.029,Y -239.744,Z 1025.726,A 0.000,B 0.000,C 90.000,E1 310.701} C_DIS
LIN {X 0.103,Y -247.361,Z 1025.716,A 0.000,B 0.000,C 90.000,E1 308.830} C_DIS
LIN {X -0.005,Y -255.906,Z 1025.706,A 0.000,B 0.000,C 90.000,E1 307.030} C_DIS
LIN {X -0.082,Y -267.358,Z 1025.694,A 0.000,B 0.000,C 90.000,E1 304.898} C_DIS
LIN {X 0.026,Y -283.961,Z 1025.678,A 0.000,B 0.000,C 90.000,E1 302.084} C_DIS
LIN {X -0.127,Y -304.152,Z 1025.661,A 0.000,B 0.000,C 90.000,E1 299.077} C_DIS
LIN {X 0.140,Y -321.145,Z 1025.649,A 0.000,B 0.000,C 90.000,E1 296.744} C_DIS
LIN {X 0.132,Y -334.136,Z 1025.640,A 0.000,B 0.000,C 90.000,E1 295.207} C_DIS
LIN {X -0.115,Y -353.076,Z 1025.629,A 0.000,B 0.000,C 90.000,E1 293.259} C_DIS
LIN {X -0.055,Y -380.624,Z 1025.615,A 0.000,B 0.000,C 90.000,E1 290.663} C_DIS
LIN {X -0.123,Y -394.294,Z 1025.608,A 0.000,B 0.000,C 90.000,E1 289.450} C_DIS
LIN {X -0.058,Y -405.154,Z 1025.603,A 0.000,B 0.000,C 90.000,E1 288.471} C_DIS
LIN {X 0.209,Y -415.700,Z 1025.597,A 0.000,B 0.000,C 90.000,E1 287.457} C_DIS
LIN {X 0.020,Y -423.258,Z 1025.593,A 0.000,B 0.000,C 90.000,E1 286.732} C_DIS
LIN {X 0.222,Y -433.095,Z 1025.587,A 0.000,B 0.000,C 90.000,E1 285.662} C_DIS
LIN {X -0.046,Y -440.208,Z 1025.583,A 0.000,B 0.000,C 90.000,E1 284.898} C_DIS
LIN {X 0.064,Y -449.129,Z 1025.577,A 0.000,B 0.000,C 90.000,E1 283.828} C_DIS
LIN {X -0.082,Y -455.371,Z 1025.573,A 0.000,B 0.000,C 90.000,E1 283.063} C_DIS
LIN {X -0.181,Y -461.081,Z 1025.568,A 0.000,B 0.000,C 90.000,E1 282.299} C_DIS
LIN {X 0.069,Y -467.890,Z 1025.563,A 0.000,B 0.000,C 90.000,E1 281.243} C_DIS
LIN {X -0.006,Y -472.343,Z 1025.558,A 0.000,B 0.000,C 90.000,E1 280.489} C_DIS
LIN {X 0.038,Y -476.199,Z 1025.554,A 0.000,B 0.000,C 90.000,E1 279.726} C_DIS
LIN {X 0.165,Y -478.476,Z 1025.551,A 0.000,B 0.000,C 90.000,E1 279.208} C_DIS
LIN {X -0.166,Y -480.455,Z 1025.548,A 0.000,B 0.000,C 90.000,E1 278.746} C_DIS
LIN {X 0.057,Y -482.204,Z 1025.546,A 0.000,B 0.000,C 90.000,E1 278.219} C_DIS
LIN {X 0.222,Y -483.676,Z 1025.543,A 0.000,B 0.000,C 90.000,E1 277.701} C_DIS
LIN {X -0.083,Y -484.948,Z 1025.540,A 0.000,B 0.000,C 90.000,E1 277.239} C_DIS
LIN {X 0.103,Y -485.997,Z 1025.537,A 0.000,B 0.000,C 90.000,E1 276.720} C_DIS
LIN {X -0.188,Y -486.838,Z 1025.535,A 0.000,B 0.000,C 90.000,E1 276.258} C_DIS
LIN {X 0.011,Y -487.406,Z 1025.532,A 0.000,B 0.000,C 90.000,E1 275.739} C_DIS
LIN {X 0.215,Y -487.612,Z 1025.529,A 0.000,B 0.000,C 90.000,E1 275.220} C_DIS
LIN {X -0.066,Y -487.372,Z 1025.526,A 0.000,B 0.000,C 90.000,E1 274.759} C_DIS
LIN {X 0.101,Y -486.658,Z 1025.524,A 0.000,B 0.000,C 90.000,E1 274.245} C_DIS
LIN {X -0.180,Y -485.426,Z 1025.521,A 0.000,B 0.000,C 90.000,E1 273.784} C_DIS
LIN {X -0.013,Y -483.603,Z 1025.518,A 0.000,B 0.000,C 90.000,E1 273.269} C_DIS
LIN {X 0.175,Y -481.086,Z 1025.515,A 0.000,B 0.000,C 90.000,E1 272.751} C_DIS
LIN {X -0.160,Y -477.864,Z 1025.513,A 0.000,B 0.000,C 90.000,E1 272.293} C_DIS
LIN {X -0.013,Y -473.787,Z 1025.510,A 0.000,B 0.000,C 90.000,E1 271.776} C_DIS
LIN {X 0.094,Y -468.805,Z 1025.507,A 0.000,B 0.000,C 90.000,E1 271.260} C_DIS
LIN {X -0.128,Y -463.046,Z 1025.504,A 0.000,B 0.000,C 90.000,E1 270.802} C_DIS
LIN {X 0.107,Y -456.989,Z 1025.502,A 0.000,B 0.000,C 90.000,E1 270.344} C_DIS
LIN {X -0.033,Y -453.889,Z 1025.501,A 0.000,B 0.000,C 90.000,E1 270.172} C_DIS
LIN {X -0.046,Y -446.997,Z 1025.499,A 0.000,B 0.000,C 90.000,E1 269.828} C_DIS
LIN {X 0.016,Y -439.549,Z 1025.497,A 0.000,B 0.000,C 90.000,E1 269.542} C_DIS
LIN {X 0.116,Y -431.704,Z 1025.496,A 0.000,B 0.000,C 90.000,E1 269.312} C_DIS
LIN {X -0.186,Y -423.020,Z 1025.495,A 0.000,B 0.000,C 90.000,E1 269.198} C_DIS
LIN {X -0.131,Y -414.184,Z 1025.495,A 0.000,B 0.000,C 90.000,E1 269.083} C_DIS
LIN {X 0.115,Y -403.209,Z 1025.494,A 0.000,B 0.000,C 90.000,E1 268.969} C_DIS
LIN {X -0.007,Y -399.054,Z 1025.494,A 0.000,B 0.000,C 90.000,E1 268.969} C_DIS
LIN {X -0.031,Y -181.310,Z 1025.494,A 0.000,B 0.000,C 90.000,E1 268.969} C_DIS
LIN {X 0.022,Y -180.900,Z 1025.474,A 0.000,B 0.000,C 90.000,E1 265.241} C_DIS
LIN {X -0.028,Y -180.220,Z 1025.464,A 0.000,B 0.000,C 90.000,E1 263.571} C_DIS
LIN {X -0.074,Y -179.037,Z 1025.445,A 0.000,B 0.000,C 90.000,E1 260.208} C_DIS
LIN {X -0.012,Y -178.699,Z 1025.441,A 0.000,B 0.000,C 90.000,E1 259.342} C_DIS
LIN {X 0.098,Y -175.748,Z 1025.412,A 0.000,B 0.000,C 90.000,E1 254.212} C_DIS
LIN {X 0.093,Y -171.933,Z 1025.384,A 0.000,B 0.000,C 90.000,E1 249.082} C_DIS
LIN {X 0.067,Y -171.310,Z 1025.379,A 0.000,B 0.000,C 90.000,E1 248.230} C_DIS
LIN {X -0.038,Y -167.570,Z 1025.355,A 0.000,B 0.000,C 90.000,E1 243.948} C_DIS
LIN {X -0.099,Y -166.200,Z 1025.346,A 0.000,B 0.000,C 90.000,E1 242.231} C_DIS
LIN {X -0.025,Y -162.967,Z 1025.326,A 0.000,B 0.000,C 90.000,E1 238.712} C_DIS
LIN {X -0.062,Y -160.877,Z 1025.312,A 0.000,B 0.000,C 90.000,E1 236.087} C_DIS
LIN {X -0.083,Y -157.650,Z 1025.292,A 0.000,B 0.000,C 90.000,E1 232.557} C_DIS
LIN {X 0.075,Y -155.687,Z 1025.277,A 0.000,B 0.000,C 90.000,E1 229.828} C_DIS
LIN {X 0.020,Y -151.953,Z 1025.252,A 0.000,B 0.000,C 90.000,E1 225.364} C_DIS
LIN {X -0.071,Y -150.191,Z 1025.237,A 0.000,B 0.000,C 90.000,E1 222.690} C_DIS
LIN {X 0.060,Y -146.964,Z 1025.212,A 0.000,B 0.000,C 90.000,E1 218.096} C_DIS
LIN {X -0.037,Y -145.551,Z 1025.197,A 0.000,B 0.000,C 90.000,E1 215.391} C_DIS
LIN {X -0.037,Y -142.944,Z 1025.171,A 0.000,B 0.000,C 90.000,E1 210.797} C_DIS
LIN {X 0.020,Y -141.569,Z 1025.151,A 0.000,B 0.000,C 90.000,E1 207.078} C_DIS
LIN {X -0.058,Y -139.412,Z 1025.114,A 0.000,B 0.000,C 90.000,E1 200.610} C_DIS
LIN {X -0.006,Y -139.134,Z 1025.104,A 0.000,B 0.000,C 90.000,E1 198.725} C_DIS
LIN {X 0.021,Y -138.350,Z 1025.057,A 0.000,B 0.000,C 90.000,E1 190.310} C_DIS
LIN {X 0.009,Y -139.495,Z 1025.005,A 0.000,B 0.000,C 90.000,E1 180.974} C_DIS
LIN {X -0.050,Y -141.112,Z 1024.974,A 0.000,B 0.000,C 90.000,E1 175.412} C_DIS
LIN {X 0.044,Y -142.492,Z 1024.959,A 0.000,B 0.000,C 90.000,E1 172.591} C_DIS
LIN {X -0.010,Y -144.745,Z 1024.933,A 0.000,B 0.000,C 90.000,E1 167.993} C_DIS
LIN {X -0.059,Y -147.352,Z 1024.913,A 0.000,B 0.000,C 90.000,E1 164.338} C_DIS
LIN {X 0.005,Y -150.677,Z 1024.888,A 0.000,B 0.000,C 90.000,E1 159.752} C_DIS
LIN {X 0.089,Y -154.157,Z 1024.867,A 0.000,B 0.000,C 90.000,E1 156.102} C_DIS
LIN {X 0.020,Y -157.588,Z 1024.847,A 0.000,B 0.000,C 90.000,E1 152.538} C_DIS
LIN {X -0.029,Y -161.836,Z 1024.828,A 0.000,B 0.000,C 90.000,E1 148.997} C_DIS
LIN {X -0.012,Y -166.027,Z 1024.808,A 0.000,B 0.000,C 90.000,E1 145.468} C_DIS
LIN {X -0.019,Y -171.029,Z 1024.789,A 0.000,B 0.000,C 90.000,E1 141.984} C_DIS
LIN {X 0.011,Y -175.900,Z 1024.770,A 0.000,B 0.000,C 90.000,E1 138.528} C_DIS
LIN {X 0.016,Y -181.503,Z 1024.751,A 0.000,B 0.000,C 90.000,E1 135.121} C_DIS
LIN {X 0.023,Y -187.022,Z 1024.732,A 0.000,B 0.000,C 90.000,E1 131.757} C_DIS
LIN {X 0.024,Y -190.140,Z 1024.723,A 0.000,B 0.000,C 90.000,E1 130.092} C_DIS
LIN {X -0.064,Y -197.056,Z 1024.701,A 0.000,B 0.000,C 90.000,E1 126.217} C_DIS
LIN {X 0.110,Y -302.016,Z 1024.701,A 0.000,B 0.000,C 90.000,E1 126.171} C_DIS
LIN {X 0.038,Y -303.165,Z 1024.701,A 0.000,B 0.000,C 90.000,E1 126.171} C_DIS
LIN {X -0.139,Y -307.964,Z 1024.700,A 0.000,B 0.000,C 90.000,E1 126.011} C_DIS
LIN {X 0.047,Y -311.047,Z 1024.698,A 0.000,B 0.000,C 90.000,E1 125.724} C_DIS
LIN {X 0.128,Y -314.760,Z 1024.696,A 0.000,B 0.000,C 90.000,E1 125.231} C_DIS
LIN {X -0.083,Y -316.523,Z 1024.694,A 0.000,B 0.000,C 90.000,E1 124.945} C_DIS
LIN {X -0.034,Y -317.904,Z 1024.692,A 0.000,B 0.000,C 90.000,E1 124.612} C_DIS
LIN {X -0.160,Y -330.127,Z 1024.673,A 0.000,B 0.000,C 90.000,E1 121.131} C_DIS
LIN {X 0.073,Y -341.542,Z 1024.657,A 0.000,B 0.000,C 90.000,E1 118.281} C_DIS
LIN {X 0.000,Y -354.377,Z 1024.642,A 0.000,B 0.000,C 90.000,E1 115.540} C_DIS
LIN {X 0.069,Y -367.074,Z 1024.629,A 0.000,B 0.000,C 90.000,E1 113.131} C_DIS
LIN {X 0.018,Y -381.075,Z 1024.615,A 0.000,B 0.000,C 90.000,E1 110.791} C_DIS
LIN {X 0.061,Y -396.478,Z 1024.603,A 0.000,B 0.000,C 90.000,E1 108.489} C_DIS
LIN {X -0.016,Y -413.394,Z 1024.590,A 0.000,B 0.000,C 90.000,E1 106.260} C_DIS
LIN {X 0.087,Y -431.944,Z 1024.578,A 0.000,B 0.000,C 90.000,E1 104.064} C_DIS
LIN {X -0.083,Y -451.825,Z 1024.567,A 0.000,B 0.000,C 90.000,E1 102.007} C_DIS
LIN {X 0.019,Y -467.119,Z 1024.559,A 0.000,B 0.000,C 90.000,E1 100.546} C_DIS
LIN {X 0.037,Y -469.226,Z 1024.557,A 0.000,B 0.000,C 90.000,E1 100.310} C_DIS
LIN {X -0.116,Y -470.945,Z 1024.556,A 0.000,B 0.000,C 90.000,E1 100.074} C_DIS
LIN {X 0.115,Y -472.235,Z 1024.554,A 0.000,B 0.000,C 90.000,E1 99.792} C_DIS
LIN {X -0.171,Y -473.839,Z 1024.552,A 0.000,B 0.000,C 90.000,E1 99.321} C_DIS
LIN {X -0.059,Y -474.388,Z 1024.549,A 0.000,B 0.000,C 90.000,E1 98.803} C_DIS
LIN {X 0.133,Y -473.972,Z 1024.546,A 0.000,B 0.000,C 90.000,E1 98.276} C_DIS
LIN {X -0.211,Y -472.534,Z 1024.543,A 0.000,B 0.000,C 90.000,E1 97.814} C_DIS
LIN {X 0.054,Y -471.358,Z 1024.542,A 0.000,B 0.000,C 90.000,E1 97.530} C_DIS
LIN {X 0.172,Y -468.018,Z 1024.539,A 0.000,B 0.000,C 90.000,E1 97.011} C_DIS
LIN {X -0.045,Y -457.473,Z 1024.531,A 0.000,B 0.000,C 90.000,E1 95.511} C_DIS
LIN {X -0.193,Y -436.340,Z 1024.513,A 0.000,B 0.000,C 90.000,E1 92.407} C_DIS
LIN {X -0.158,Y -422.025,Z 1024.500,A 0.000,B 0.000,C 90.000,E1 90.000} C_DIS
LIN {X -0.078,Y -408.841,Z 1024.486,A 0.000,B 0.000,C 90.000,E1 87.535} C_DIS
LIN {X -0.055,Y -399.924,Z 1024.477,A 0.000,B 0.000,C 90.000,E1 85.869} C_DIS
LIN {X -0.191,Y -390.857,Z 1024.468,A 0.000,B 0.000,C 90.000,E1 84.204} C_DIS
LIN {X -0.044,Y -380.009,Z 1024.457,A 0.000,B 0.000,C 90.000,E1 82.186} C_DIS
LIN {X -0.022,Y -370.314,Z 1024.447,A 0.000,B 0.000,C 90.000,E1 80.443} C_DIS
LIN {X -0.173,Y -360.381,Z 1024.437,A 0.000,B 0.000,C 90.000,E1 78.701} C_DIS
LIN {X -0.076,Y -348.757,Z 1024.425,A 0.000,B 0.000,C 90.000,E1 76.589} C_DIS
LIN {X 0.153,Y -334.209,Z 1024.410,A 0.000,B 0.000,C 90.000,E1 73.795} C_DIS
LIN {X -0.083,Y -321.660,Z 1024.396,A 0.000,B 0.000,C 90.000,E1 71.329} C_DIS
LIN {X -0.029,Y -311.019,Z 1024.384,A 0.000,B 0.000,C 90.000,E1 69.082} C_DIS
LIN {X 0.066,Y -297.708,Z 1024.367,A 0.000,B 0.000,C 90.000,E1 66.125} C_DIS
LIN {X 0.024,Y -286.154,Z 1024.353,A 0.000,B 0.000,C 90.000,E1 63.461} C_DIS
LIN {X 0.091,Y -274.856,Z 1024.337,A 0.000,B 0.000,C 90.000,E1 60.717} C_DIS
LIN {X -0.133,Y -265.142,Z 1024.324,A 0.000,B 0.000,C 90.000,E1 58.329} C_DIS
LIN {X -0.002,Y -252.979,Z 1024.306,A 0.000,B 0.000,C 90.000,E1 55.102} C_DIS
LIN {X 0.010,Y -241.428,Z 1024.288,A 0.000,B 0.000,C 90.000,E1 51.823} C_DIS
LIN {X -0.039,Y -230.645,Z 1024.269,A 0.000,B 0.000,C 90.000,E1 48.485} C_DIS
LIN {X 0.117,Y -221.595,Z 1024.252,A 0.000,B 0.000,C 90.000,E1 45.405} C_DIS
LIN {X -0.085,Y -212.939,Z 1024.235,A 0.000,B 0.000,C 90.000,E1 42.366} C_DIS
LIN {X -0.002,Y -204.788,Z 1024.218,A 0.000,B 0.000,C 90.000,E1 39.197} C_DIS
LIN {X -0.061,Y -197.262,Z 1024.200,A 0.000,B 0.000,C 90.000,E1 36.011} C_DIS
LIN {X -0.052,Y -190.339,Z 1024.182,A 0.000,B 0.000,C 90.000,E1 32.752} C_DIS
LIN {X 0.064,Y -184.210,Z 1024.163,A 0.000,B 0.000,C 90.000,E1 29.411} C_DIS
LIN {X -0.077,Y -178.884,Z 1024.145,A 0.000,B 0.000,C 90.000,E1 26.104} C_DIS
LIN {X -0.023,Y -174.389,Z 1024.126,A 0.000,B 0.000,C 90.000,E1 22.695} C_DIS
LIN {X -0.054,Y -169.745,Z 1024.102,A 0.000,B 0.000,C 90.000,E1 18.417} C_DIS
LIN {X 0.004,Y -166.204,Z 1024.078,A 0.000,B 0.000,C 90.000,E1 14.064} C_DIS
LIN {X 0.051,Y -163.418,Z 1024.049,A 0.000,B 0.000,C 90.000,E1 8.803} C_DIS
LIN {X 0.020,Y -164.182,Z 1023.953,A 0.000,B 0.000,C 90.000,E1 351.602} C_DIS
LIN {X 0.007,Y -166.779,Z 1023.929,A 0.000,B 0.000,C 90.000,E1 347.229} C_DIS
LIN {X -0.071,Y -170.359,Z 1023.905,A 0.000,B 0.000,C 90.000,E1 342.906} C_DIS
LIN {X -0.044,Y -174.008,Z 1023.886,A 0.000,B 0.000,C 90.000,E1 339.444} C_DIS
LIN {X 0.035,Y -178.480,Z 1023.867,A 0.000,B 0.000,C 90.000,E1 335.997} C_DIS
LIN {X 0.023,Y -183.788,Z 1023.848,A 0.000,B 0.000,C 90.000,E1 332.615} C_DIS
LIN {X -0.011,Y -189.928,Z 1023.829,A 0.000,B 0.000,C 90.000,E1 329.282} C_DIS
LIN {X -0.092,Y -196.781,Z 1023.811,A 0.000,B 0.000,C 90.000,E1 326.008} C_DIS
LIN {X -0.064,Y -205.238,Z 1023.791,A 0.000,B 0.000,C 90.000,E1 322.351} C_DIS
LIN {X 0.051,Y -213.300,Z 1023.773,A 0.000,B 0.000,C 90.000,E1 319.138} C_DIS
LIN {X -0.029,Y -223.178,Z 1023.754,A 0.000,B 0.000,C 90.000,E1 315.648} C_DIS
LIN {X -0.106,Y -232.879,Z 1023.737,A 0.000,B 0.000,C 90.000,E1 312.609} C_DIS
LIN {X 0.011,Y -239.706,Z 1023.726,A 0.000,B 0.000,C 90.000,E1 310.701} C_DIS
LIN {X 0.084,Y -247.317,Z 1023.716,A 0.000,B 0.000,C 90.000,E1 308.830} C_DIS
LIN {X -0.024,Y -255.884,Z 1023.706,A 0.000,B 0.000,C 90.000,E1 307.030} C_DIS
LIN {X -0.103,Y -267.344,Z 1023.694,A 0.000,B 0.000,C 90.000,E1 304.898} C_DIS
LIN {X -0.043,Y -286.159,Z 1023.676,A 0.000,B 0.000,C 90.000,E1 301.750} C_DIS
LIN {X -0.129,Y -306.557,Z 1023.660,A 0.000,B 0.000,C 90.000,E1 298.743} C_DIS
LIN {X 0.118,Y -321.247,Z 1023.649,A 0.000,B 0.000,C 90.000,E1 296.744} C_DIS
LIN {X 0.204,Y -334.149,Z 1023.640,A 0.000,B 0.000,C 90.000,E1 295.207} C_DIS
LIN {X -0.044,Y -355.681,Z 1023.628,A 0.000,B 0.000,C 90.000,E1 293.003} C_DIS
LIN {X -0.017,Y -383.300,Z 1023.613,A 0.000,B 0.000,C 90.000,E1 290.429} C_DIS
LIN {X 0.003,Y -399.674,Z 1023.605,A 0.000,B 0.000,C 90.000,E1 288.960} C_DIS
LIN {X -0.063,Y -410.332,Z 1023.600,A 0.000,B 0.000,C 90.000,E1 288.000} C_DIS
LIN {X 0.195,Y -418.156,Z 1023.596,A 0.000,B 0.000,C 90.000,E1 287.221} C_DIS
LIN {X -0.105,Y -425.685,Z 1023.592,A 0.000,B 0.000,C 90.000,E1 286.496} C_DIS
LIN {X -0.033,Y -435.494,Z 1023.586,A 0.000,B 0.000,C 90.000,E1 285.426} C_DIS
LIN {X 0.020,Y -444.714,Z 1023.580,A 0.000,B 0.000,C 90.000,E1 284.356} C_DIS
LIN {X 0.074,Y -453.296,Z 1023.574,A 0.000,B 0.000,C 90.000,E1 283.300} C_DIS
LIN {X -0.035,Y -459.224,Z 1023.570,A 0.000,B 0.000,C 90.000,E1 282.535} C_DIS
LIN {X 0.197,Y -466.259,Z 1023.564,A 0.000,B 0.000,C 90.000,E1 281.478} C_DIS
LIN {X 0.103,Y -470.920,Z 1023.560,A 0.000,B 0.000,C 90.000,E1 280.725} C_DIS
LIN {X 0.143,Y -475.006,Z 1023.555,A 0.000,B 0.000,C 90.000,E1 279.962} C_DIS
LIN {X 0.131,Y -478.519,Z 1023.551,A 0.000,B 0.000,C 90.000,E1 279.208} C_DIS
LIN {X -0.200,Y -480.520,Z 1023.548,A 0.000,B 0.000,C 90.000,E1 278.746} C_DIS
LIN {X 0.023,Y -482.270,Z 1023.546,A 0.000,B 0.000,C 90.000,E1 278.219} C_DIS
LIN {X 0.187,Y -483.747,Z 1023.543,A 0.000,B 0.000,C 90.000,E1 277.701} C_DIS
LIN {X -0.117,Y -485.033,Z 1023.540,A 0.000,B 0.000,C 90.000,E1 277.239} C_DIS
LIN {X 0.068,Y -486.099,Z 1023.537,A 0.000,B 0.000,C 90.000,E1 276.720} C_DIS
LIN {X -0.221,Y -486.960,Z 1023.535,A 0.000,B 0.000,C 90.000,E1 276.258} C_DIS
LIN {X -0.021,Y -487.548,Z 1023.532,A 0.000,B 0.000,C 90.000,E1 275.739} C_DIS
LIN {X 0.183,Y -487.769,Z 1023.529,A 0.000,B 0.000,C 90.000,E1 275.220} C_DIS
LIN {X -0.097,Y -487.535,Z 1023.526,A 0.000,B 0.000,C 90.000,E1 274.759} C_DIS
LIN {X 0.071,Y -486.821,Z 1023.524,A 0.000,B 0.000,C 90.000,E1 274.245} C_DIS
LIN {X -0.209,Y -485.598,Z 1023.521,A 0.000,B 0.000,C 90.000,E1 273.784} C_DIS
LIN {X -0.041,Y -483.793,Z 1023.518,A 0.000,B 0.000,C 90.000,E1 273.269} C_DIS
LIN {X 0.147,Y -481.338,Z 1023.515,A 0.000,B 0.000,C 90.000,E1 272.751} C_DIS
LIN {X -0.186,Y -478.094,Z 1023.513,A 0.000,B 0.000,C 90.000,E1 272.293} C_DIS
LIN {X -0.037,Y -474.072,Z 1023.510,A 0.000,B 0.000,C 90.000,E1 271.776} C_DIS
LIN {X 0.072,Y -469.119,Z 1023.507,A 0.000,B 0.000,C 90.000,E1 271.260} C_DIS
LIN {X -0.159,Y -463.376,Z 1023.504,A 0.000,B 0.000,C 90.000,E1 270.802} C_DIS
LIN {X 0.065,Y -457.261,Z 1023.502,A 0.000,B 0.000,C 90.000,E1 270.344} C_DIS
LIN {X -0.068,Y -454.176,Z 1023.501,A 0.000,B 0.000,C 90.000,E1 270.172} C_DIS
LIN {X -0.080,Y -447.284,Z 1023.499,A 0.000,B 0.000,C 90.000,E1 269.828} C_DIS
LIN {X -0.033,Y -439.874,Z 1023.497,A 0.000,B 0.000,C 90.000,E1 269.542} C_DIS
LIN {X 0.060,Y -432.120,Z 1023.496,A 0.000,B 0.000,C 90.000,E1 269.312} C_DIS
LIN {X 0.186,Y -423.559,Z 1023.495,A 0.000,B 0.000,C 90.000,E1 269.141} C_DIS
LIN {X -0.185,Y -414.621,Z 1023.495,A 0.000,B 0.000,C 90.000,E1 269.083} C_DIS
LIN {X 0.041,Y -403.770,Z 1023.494,A 0.000,B 0.000,C 90.000,E1 268.969} C_DIS
LIN {X -0.090,Y -399.755,Z 1023.494,A 0.000,B 0.000,C 90.000,E1 268.969} C_DIS
LIN {X -0.070,Y -181.307,Z 1023.494,A 0.000,B 0.000,C 90.000,E1 268.969} C_DIS
LIN {X -0.019,Y -180.899,Z 1023.474,A 0.000,B 0.000,C 90.000,E1 265.241} C_DIS
LIN {X -0.069,Y -180.215,Z 1023.464,A 0.000,B 0.000,C 90.000,E1 263.571} C_DIS
LIN {X 0.061,Y -179.034,Z 1023.445,A 0.000,B 0.000,C 90.000,E1 260.151} C_DIS
LIN {X -0.053,Y -178.692,Z 1023.441,A 0.000,B 0.000,C 90.000,E1 259.342} C_DIS
LIN {X 0.057,Y -175.740,Z 1023.412,A 0.000,B 0.000,C 90.000,E1 254.212} C_DIS
LIN {X 0.053,Y -171.925,Z 1023.384,A 0.000,B 0.000,C 90.000,E1 249.082} C_DIS
LIN {X 0.028,Y -171.298,Z 1023.379,A 0.000,B 0.000,C 90.000,E1 248.230} C_DIS
LIN {X 0.073,Y -167.560,Z 1023.355,A 0.000,B 0.000,C 90.000,E1 243.896} C_DIS
LIN {X 0.086,Y -166.186,Z 1023.345,A 0.000,B 0.000,C 90.000,E1 242.153} C_DIS
LIN {X 0.076,Y -162.955,Z 1023.326,A 0.000,B 0.000,C 90.000,E1 238.663} C_DIS
LIN {X -0.100,Y -160.863,Z 1023.311,A 0.000,B 0.000,C 90.000,E1 236.087} C_DIS
LIN {X 0.100,Y -157.638,Z 1023.292,A 0.000,B 0.000,C 90.000,E1 232.477} C_DIS
LIN {X 0.038,Y -155.676,Z 1023.277,A 0.000,B 0.000,C 90.000,E1 229.828} C_DIS
LIN {X -0.017,Y -151.942,Z 1023.252,A 0.000,B 0.000,C 90.000,E1 225.364} C_DIS
LIN {X -0.006,Y -150.181,Z 1023.237,A 0.000,B 0.000,C 90.000,E1 222.651} C_DIS
LIN {X 0.023,Y -146.955,Z 1023.212,A 0.000,B 0.000,C 90.000,E1 218.096} C_DIS
LIN {X 0.011,Y -145.542,Z 1023.196,A 0.000,B 0.000,C 90.000,E1 215.358} C_DIS
LIN {X -0.072,Y -142.938,Z 1023.171,A 0.000,B 0.000,C 90.000,E1 210.797} C_DIS
LIN {X -0.015,Y -141.562,Z 1023.150,A 0.000,B 0.000,C 90.000,E1 207.078} C_DIS
LIN {X 0.037,Y -139.409,Z 1023.114,A 0.000,B 0.000,C 90.000,E1 200.556} C_DIS
LIN {X -0.041,Y -139.131,Z 1023.104,A 0.000,B 0.000,C 90.000,E1 198.725} C_DIS
LIN {X -0.014,Y -138.350,Z 1023.057,A 0.000,B 0.000,C 90.000,E1 190.310} C_DIS
LIN {X -0.026,Y -139.498,Z 1023.005,A 0.000,B 0.000,C 90.000,E1 180.974} C_DIS
LIN {X 0.054,Y -141.118,Z 1022.974,A 0.000,B 0.000,C 90.000,E1 175.355} C_DIS
LIN {X 0.008,Y -142.499,Z 1022.959,A 0.000,B 0.000,C 90.000,E1 172.591} C_DIS
LIN {X -0.046,Y -144.753,Z 1022.933,A 0.000,B 0.000,C 90.000,E1 167.993} C_DIS
LIN {X 0.046,Y -147.362,Z 1022.913,A 0.000,B 0.000,C 90.000,E1 164.283} C_DIS
LIN {X -0.032,Y -150.689,Z 1022.887,A 0.000,B 0.000,C 90.000,E1 159.752} C_DIS
LIN {X 0.051,Y -154.169,Z 1022.867,A 0.000,B 0.000,C 90.000,E1 156.102} C_DIS
LIN {X -0.018,Y -157.603,Z 1022.847,A 0.000,B 0.000,C 90.000,E1 152.538} C_DIS
LIN {X -0.068,Y -161.855,Z 1022.828,A 0.000,B 0.000,C 90.000,E1 148.997} C_DIS
LIN {X -0.050,Y -166.045,Z 1022.808,A 0.000,B 0.000,C 90.000,E1 145.468} C_DIS
LIN {X -0.060,Y -171.049,Z 1022.789,A 0.000,B 0.000,C 90.000,E1 141.984} C_DIS
LIN {X -0.029,Y -175.920,Z 1022.770,A 0.000,B 0.000,C 90.000,E1 138.528} C_DIS
LIN {X -0.037,Y -180.159,Z 1022.755,A 0.000,B 0.000,C 90.000,E1 135.972} C_DIS
LIN {X -0.068,Y -185.576,Z 1022.737,A 0.000,B 0.000,C 90.000,E1 132.609} C_DIS
LIN {X -0.018,Y -190.165,Z 1022.723,A 0.000,B 0.000,C 90.000,E1 130.092} C_DIS
LIN {X 0.090,Y -196.970,Z 1022.701,A 0.000,B 0.000,C 90.000,E1 126.217} C_DIS
LIN {X 0.092,Y -301.798,Z 1022.701,A 0.000,B 0.000,C 90.000,E1 126.217} C_DIS
LIN {X 0.046,Y -302.671,Z 1022.701,A 0.000,B 0.000,C 90.000,E1 126.217} C_DIS
LIN {X 0.042,Y -308.597,Z 1022.700,A 0.000,B 0.000,C 90.000,E1 125.964} C_DIS
LIN {X -0.104,Y -311.546,Z 1022.698,A 0.000,B 0.000,C 90.000,E1 125.724} C_DIS
LIN {X 0.003,Y -315.256,Z 1022.695,A 0.000,B 0.000,C 90.000,E1 125.185} C_DIS
LIN {X -0.025,Y -316.875,Z 1022.694,A 0.000,B 0.000,C 90.000,E1 124.865} C_DIS
LIN {X 0.094,Y -319.195,Z 1022.690,A 0.000,B 0.000,C 90.000,E1 124.199} C_DIS
LIN {X -0.095,Y -330.361,Z 1022.672,A 0.000,B 0.000,C 90.000,E1 121.052} C_DIS
LIN {X -0.022,Y -341.809,Z 1022.657,A 0.000,B 0.000,C 90.000,E1 118.231} C_DIS
LIN {X 0.070,Y -354.680,Z 1022.642,A 0.000,B 0.000,C 90.000,E1 115.463} C_DIS
LIN {X -0.003,Y -367.411,Z 1022.628,A 0.000,B 0.000,C 90.000,E1 113.078} C_DIS
LIN {X -0.041,Y -381.448,Z 1022.615,A 0.000,B 0.000,C 90.000,E1 110.737} C_DIS
LIN {X 0.139,Y -396.889,Z 1022.602,A 0.000,B 0.000,C 90.000,E1 108.417} C_DIS
LIN {X -0.051,Y -413.848,Z 1022.590,A 0.000,B 0.000,C 90.000,E1 106.205} C_DIS
LIN {X 0.067,Y -432.443,Z 1022.578,A 0.000,B 0.000,C 90.000,E1 104.008} C_DIS
LIN {X -0.067,Y -452.344,Z 1022.566,A 0.000,B 0.000,C 90.000,E1 101.951} C_DIS
LIN {X 0.065,Y -467.604,Z 1022.558,A 0.000,B 0.000,C 90.000,E1 100.489} C_DIS
LIN {X 0.087,Y -469.585,Z 1022.557,A 0.000,B 0.000,C 90.000,E1 100.254} C_DIS
LIN {X -0.064,Y -471.213,Z 1022.556,A 0.000,B 0.000,C 90.000,E1 100.018} C_DIS
LIN {X 0.249,Y -472.434,Z 1022.554,A 0.000,B 0.000,C 90.000,E1 99.726} C_DIS
LIN {X -0.115,Y -473.930,Z 1022.551,A 0.000,B 0.000,C 90.000,E1 99.265} C_DIS
LIN {X -0.001,Y -474.386,Z 1022.549,A 0.000,B 0.000,C 90.000,E1 98.746} C_DIS
LIN {X 0.192,Y -473.881,Z 1022.546,A 0.000,B 0.000,C 90.000,E1 98.219} C_DIS
LIN {X -0.151,Y -472.337,Z 1022.543,A 0.000,B 0.000,C 90.000,E1 97.757} C_DIS
LIN {X 0.114,Y -471.095,Z 1022.542,A 0.000,B 0.000,C 90.000,E1 97.473} C_DIS
LIN {X 0.169,Y -462.448,Z 1022.535,A 0.000,B 0.000,C 90.000,E1 96.201} C_DIS
LIN {X -0.147,Y -451.750,Z 1022.526,A 0.000,B 0.000,C 90.000,E1 94.702} C_DIS
LIN {X -0.151,Y -436.068,Z 1022.513,A 0.000,B 0.000,C 90.000,E1 92.350} C_DIS
LIN {X 0.172,Y -423.271,Z 1022.501,A 0.000,B 0.000,C 90.000,E1 90.172} C_DIS
LIN {X -0.130,Y -410.045,Z 1022.487,A 0.000,B 0.000,C 90.000,E1 87.764} C_DIS
LIN {X -0.110,Y -401.162,Z 1022.478,A 0.000,B 0.000,C 90.000,E1 86.102} C_DIS
LIN {X 0.198,Y -392.107,Z 1022.469,A 0.000,B 0.000,C 90.000,E1 84.375} C_DIS
LIN {X -0.017,Y -381.262,Z 1022.458,A 0.000,B 0.000,C 90.000,E1 82.413} C_DIS
LIN {X 0.016,Y -374.902,Z 1022.451,A 0.000,B 0.000,C 90.000,E1 81.254} C_DIS
LIN {X -0.050,Y -365.054,Z 1022.442,A 0.000,B 0.000,C 90.000,E1 79.511} C_DIS
LIN {X 0.081,Y -353.422,Z 1022.430,A 0.000,B 0.000,C 90.000,E1 77.409} C_DIS
LIN {X 0.015,Y -338.683,Z 1022.415,A 0.000,B 0.000,C 90.000,E1 74.685} C_DIS
LIN {X 0.105,Y -326.058,Z 1022.401,A 0.000,B 0.000,C 90.000,E1 72.181} C_DIS
LIN {X 0.071,Y -313.798,Z 1022.387,A 0.000,B 0.000,C 90.000,E1 69.645} C_DIS
LIN {X -0.041,Y -300.372,Z 1022.371,A 0.000,B 0.000,C 90.000,E1 66.741} C_DIS
LIN {X 0.003,Y -290.146,Z 1022.358,A 0.000,B 0.000,C 90.000,E1 64.409} C_DIS
LIN {X 0.083,Y -280.210,Z 1022.345,A 0.000,B 0.000,C 90.000,E1 62.025} C_DIS
LIN {X 0.069,Y -270.412,Z 1022.331,A 0.000,B 0.000,C 90.000,E1 59.616} C_DIS
LIN {X 0.028,Y -260.746,Z 1022.318,A 0.000,B 0.000,C 90.000,E1 57.168} C_DIS
LIN {X -0.051,Y -250.085,Z 1022.302,A 0.000,B 0.000,C 90.000,E1 54.322} C_DIS
LIN {X 0.031,Y -238.691,Z 1022.283,A 0.000,B 0.000,C 90.000,E1 51.009} C_DIS
LIN {X 0.103,Y -229.245,Z 1022.267,A 0.000,B 0.000,C 90.000,E1 48.000} C_DIS
LIN {X -0.010,Y -219.169,Z 1022.248,A 0.000,B 0.000,C 90.000,E1 44.595} C_DIS
LIN {X 0.052,Y -210.576,Z 1022.230,A 0.000,B 0.000,C 90.000,E1 41.472} C_DIS
LIN {X 0.072,Y -202.569,Z 1022.213,A 0.000,B 0.000,C 90.000,E1 38.302} C_DIS
LIN {X -0.003,Y -195.191,Z 1022.195,A 0.000,B 0.000,C 90.000,E1 35.105} C_DIS
LIN {X 0.112,Y -188.463,Z 1022.177,A 0.000,B 0.000,C 90.000,E1 31.799} C_DIS
LIN {X 0.084,Y -182.601,Z 1022.158,A 0.000,B 0.000,C 90.000,E1 28.487} C_DIS
LIN {X -0.018,Y -177.473,Z 1022.140,A 0.000,B 0.000,C 90.000,E1 25.155} C_DIS
LIN {X -0.069,Y -173.222,Z 1022.121,A 0.000,B 0.000,C 90.000,E1 21.770} C_DIS
LIN {X 0.007,Y -169.597,Z 1022.102,A 0.000,B 0.000,C 90.000,E1 18.308} C_DIS
LIN {X -0.096,Y -166.075,Z 1022.078,A 0.000,B 0.000,C 90.000,E1 14.008} C_DIS
LIN {X -0.047,Y -163.326,Z 1022.049,A 0.000,B 0.000,C 90.000,E1 8.746} C_DIS
LIN {X 0.018,Y -164.134,Z 1021.953,A 0.000,B 0.000,C 90.000,E1 351.602} C_DIS
LIN {X 0.013,Y -167.354,Z 1021.924,A 0.000,B 0.000,C 90.000,E1 346.353} C_DIS
LIN {X 0.043,Y -171.135,Z 1021.900,A 0.000,B 0.000,C 90.000,E1 342.000} C_DIS
LIN {X -0.072,Y -175.005,Z 1021.881,A 0.000,B 0.000,C 90.000,E1 338.592} C_DIS
LIN {X 0.007,Y -179.714,Z 1021.862,A 0.000,B 0.000,C 90.000,E1 335.153} C_DIS
LIN {X 0.033,Y -185.255,Z 1021.843,A 0.000,B 0.000,C 90.000,E1 331.769} C_DIS
LIN {X -0.032,Y -191.576,Z 1021.825,A 0.000,B 0.000,C 90.000,E1 328.456} C_DIS
LIN {X -0.068,Y -198.584,Z 1021.806,A 0.000,B 0.000,C 90.000,E1 325.182} C_DIS
LIN {X -0.030,Y -207.189,Z 1021.786,A 0.000,B 0.000,C 90.000,E1 321.537} C_DIS
LIN {X 0.047,Y -216.484,Z 1021.766,A 0.000,B 0.000,C 90.000,E1 317.957} C_DIS
LIN {X 0.117,Y -225.478,Z 1021.749,A 0.000,B 0.000,C 90.000,E1 314.838} C_DIS
LIN {X -0.056,Y -235.459,Z 1021.732,A 0.000,B 0.000,C 90.000,E1 311.838} C_DIS
LIN {X 0.087,Y -244.130,Z 1021.720,A 0.000,B 0.000,C 90.000,E1 309.564} C_DIS
LIN {X 0.070,Y -250.600,Z 1021.712,A 0.000,B 0.000,C 90.000,E1 308.096} C_DIS
LIN {X 0.013,Y -259.565,Z 1021.702,A 0.000,B 0.000,C 90.000,E1 306.297} C_DIS
LIN {X 0.068,Y -275.515,Z 1021.686,A 0.000,B 0.000,C 90.000,E1 303.452} C_DIS
LIN {X 0.001,Y -292.796,Z 1021.671,A 0.000,B 0.000,C 90.000,E1 300.718} C_DIS
LIN {X 0.073,Y -313.837,Z 1021.654,A 0.000,B 0.000,C 90.000,E1 297.719} C_DIS
LIN {X 0.140,Y -326.536,Z 1021.645,A 0.000,B 0.000,C 90.000,E1 296.104} C_DIS
LIN {X -0.064,Y -345.185,Z 1021.634,A 0.000,B 0.000,C 90.000,E1 294.079} C_DIS
LIN {X 0.141,Y -366.994,Z 1021.622,A 0.000,B 0.000,C 90.000,E1 291.897} C_DIS
LIN {X -0.103,Y -383.549,Z 1021.613,A 0.000,B 0.000,C 90.000,E1 290.429} C_DIS
LIN {X 0.110,Y -402.227,Z 1021.604,A 0.000,B 0.000,C 90.000,E1 288.725} C_DIS
LIN {X 0.025,Y -412.739,Z 1021.599,A 0.000,B 0.000,C 90.000,E1 287.764} C_DIS
LIN {X -0.050,Y -420.310,Z 1021.595,A 0.000,B 0.000,C 90.000,E1 287.040} C_DIS
LIN {X -0.089,Y -430.046,Z 1021.589,A 0.000,B 0.000,C 90.000,E1 286.024} C_DIS
LIN {X 0.156,Y -437.312,Z 1021.584,A 0.000,B 0.000,C 90.000,E1 285.190} C_DIS
LIN {X 0.233,Y -446.396,Z 1021.579,A 0.000,B 0.000,C 90.000,E1 284.120} C_DIS
LIN {X -0.131,Y -454.863,Z 1021.573,A 0.000,B 0.000,C 90.000,E1 283.119} C_DIS
LIN {X 0.213,Y -460.608,Z 1021.568,A 0.000,B 0.000,C 90.000,E1 282.299} C_DIS
LIN {X 0.168,Y -465.877,Z 1021.564,A 0.000,B 0.000,C 90.000,E1 281.535} C_DIS
LIN {X 0.070,Y -470.607,Z 1021.560,A 0.000,B 0.000,C 90.000,E1 280.782} C_DIS
LIN {X 0.105,Y -474.759,Z 1021.556,A 0.000,B 0.000,C 90.000,E1 280.018} C_DIS
LIN {X 0.089,Y -478.298,Z 1021.552,A 0.000,B 0.000,C 90.000,E1 279.265} C_DIS
LIN {X -0.243,Y -480.386,Z 1021.549,A 0.000,B 0.000,C 90.000,E1 278.803} C_DIS
LIN {X -0.016,Y -482.139,Z 1021.546,A 0.000,B 0.000,C 90.000,E1 278.276} C_DIS
LIN {X 0.146,Y -483.663,Z 1021.543,A 0.000,B 0.000,C 90.000,E1 277.757} C_DIS
LIN {X -0.159,Y -484.988,Z 1021.540,A 0.000,B 0.000,C 90.000,E1 277.296} C_DIS
LIN {X 0.025,Y -486.094,Z 1021.538,A 0.000,B 0.000,C 90.000,E1 276.777} C_DIS
LIN {X 0.219,Y -486.981,Z 1021.535,A 0.000,B 0.000,C 90.000,E1 276.258} C_DIS
LIN {X -0.066,Y -487.606,Z 1021.532,A 0.000,B 0.000,C 90.000,E1 275.796} C_DIS
LIN {X 0.138,Y -487.876,Z 1021.529,A 0.000,B 0.000,C 90.000,E1 275.277} C_DIS
LIN {X -0.183,Y -487.709,Z 1021.527,A 0.000,B 0.000,C 90.000,E1 274.821} C_DIS
LIN {X 0.027,Y -487.098,Z 1021.524,A 0.000,B 0.000,C 90.000,E1 274.302} C_DIS
LIN {X 0.231,Y -485.956,Z 1021.521,A 0.000,B 0.000,C 90.000,E1 273.784} C_DIS
LIN {X -0.084,Y -484.185,Z 1021.518,A 0.000,B 0.000,C 90.000,E1 273.326} C_DIS
LIN {X -0.216,Y -483.121,Z 1021.517,A 0.000,B 0.000,C 90.000,E1 273.094} C_DIS
LIN {X -0.059,Y -480.401,Z 1021.514,A 0.000,B 0.000,C 90.000,E1 272.579} C_DIS
LIN {X 0.084,Y -476.899,Z 1021.512,A 0.000,B 0.000,C 90.000,E1 272.064} C_DIS
LIN {X 0.222,Y -472.542,Z 1021.509,A 0.000,B 0.000,C 90.000,E1 271.547} C_DIS
LIN {X -0.098,Y -467.289,Z 1021.506,A 0.000,B 0.000,C 90.000,E1 271.088} C_DIS
LIN {X -0.167,Y -461.412,Z 1021.503,A 0.000,B 0.000,C 90.000,E1 270.630} C_DIS
LIN {X 0.192,Y -455.087,Z 1021.501,A 0.000,B 0.000,C 90.000,E1 270.172} C_DIS
LIN {X 0.103,Y -448.248,Z 1021.499,A 0.000,B 0.000,C 90.000,E1 269.828} C_DIS
LIN {X 0.090,Y -440.845,Z 1021.497,A 0.000,B 0.000,C 90.000,E1 269.542} C_DIS
LIN {X 0.143,Y -433.203,Z 1021.496,A 0.000,B 0.000,C 90.000,E1 269.312} C_DIS
LIN {X -0.210,Y -424.755,Z 1021.495,A 0.000,B 0.000,C 90.000,E1 269.198} C_DIS
LIN {X -0.200,Y -415.879,Z 1021.495,A 0.000,B 0.000,C 90.000,E1 269.083} C_DIS
LIN {X 0.004,Y -405.488,Z 1021.494,A 0.000,B 0.000,C 90.000,E1 268.969} C_DIS
LIN {X -0.197,Y -398.172,Z 1021.494,A 0.000,B 0.000,C 90.000,E1 268.969} C_DIS
LIN {X 0.061,Y -181.304,Z 1021.494,A 0.000,B 0.000,C 90.000,E1 268.912} C_DIS
LIN {X -0.069,Y -180.897,Z 1021.473,A 0.000,B 0.000,C 90.000,E1 265.241} C_DIS
LIN {X -0.046,Y -179.848,Z 1021.459,A 0.000,B 0.000,C 90.000,E1 262.704} C_DIS
LIN {X 0.011,Y -179.029,Z 1021.445,A 0.000,B 0.000,C 90.000,E1 260.151} C_DIS
LIN {X 0.073,Y -178.681,Z 1021.441,A 0.000,B 0.000,C 90.000,E1 259.285} C_DIS
LIN {X 0.009,Y -175.731,Z 1021.412,A 0.000,B 0.000,C 90.000,E1 254.212} C_DIS
LIN {X 0.005,Y -171.915,Z 1021.384,A 0.000,B 0.000,C 90.000,E1 249.082} C_DIS
LIN {X -0.021,Y -171.282,Z 1021.379,A 0.000,B 0.000,C 90.000,E1 248.230} C_DIS
LIN {X 0.025,Y -167.549,Z 1021.355,A 0.000,B 0.000,C 90.000,E1 243.896} C_DIS
LIN {X 0.039,Y -166.169,Z 1021.345,A 0.000,B 0.000,C 90.000,E1 242.153} C_DIS
LIN {X 0.029,Y -162.942,Z 1021.326,A 0.000,B 0.000,C 90.000,E1 238.663} C_DIS
LIN {X 0.006,Y -161.612,Z 1021.316,A 0.000,B 0.000,C 90.000,E1 236.914} C_DIS
LIN {X -0.018,Y -159.139,Z 1021.302,A 0.000,B 0.000,C 90.000,E1 234.276} C_DIS
LIN {X -0.007,Y -155.661,Z 1021.277,A 0.000,B 0.000,C 90.000,E1 229.828} C_DIS
LIN {X 0.045,Y -151.931,Z 1021.252,A 0.000,B 0.000,C 90.000,E1 225.324} C_DIS
LIN {X 0.059,Y -150.166,Z 1021.237,A 0.000,B 0.000,C 90.000,E1 222.609} C_DIS
LIN {X -0.021,Y -146.945,Z 1021.212,A 0.000,B 0.000,C 90.000,E1 218.096} C_DIS
LIN {X -0.032,Y -145.533,Z 1021.196,A 0.000,B 0.000,C 90.000,E1 215.358} C_DIS
LIN {X 0.007,Y -142.930,Z 1021.171,A 0.000,B 0.000,C 90.000,E1 210.747} C_DIS
LIN {X 0.006,Y -141.553,Z 1021.150,A 0.000,B 0.000,C 90.000,E1 207.052} C_DIS
LIN {X -0.005,Y -139.406,Z 1021.114,A 0.000,B 0.000,C 90.000,E1 200.556} C_DIS
LIN {X 0.049,Y -139.126,Z 1021.104,A 0.000,B 0.000,C 90.000,E1 198.671} C_DIS
LIN {X -0.056,Y -138.351,Z 1021.057,A 0.000,B 0.000,C 90.000,E1 190.310} C_DIS
LIN {X -0.069,Y -139.500,Z 1021.005,A 0.000,B 0.000,C 90.000,E1 180.974} C_DIS
LIN {X 0.012,Y -141.125,Z 1020.974,A 0.000,B 0.000,C 90.000,E1 175.355} C_DIS
LIN {X -0.035,Y -142.506,Z 1020.959,A 0.000,B 0.000,C 90.000,E1 172.591} C_DIS
LIN {X 0.052,Y -144.764,Z 1020.933,A 0.000,B 0.000,C 90.000,E1 167.937} C_DIS
LIN {X 0.001,Y -147.375,Z 1020.913,A 0.000,B 0.000,C 90.000,E1 164.283} C_DIS
LIN {X 0.065,Y -150.704,Z 1020.887,A 0.000,B 0.000,C 90.000,E1 159.699} C_DIS
LIN {X 0.005,Y -154.185,Z 1020.867,A 0.000,B 0.000,C 90.000,E1 156.102} C_DIS
LIN {X 0.075,Y -157.620,Z 1020.847,A 0.000,B 0.000,C 90.000,E1 152.487} C_DIS
LIN {X 0.024,Y -161.876,Z 1020.828,A 0.000,B 0.000,C 90.000,E1 148.948} C_DIS
LIN {X -0.004,Y -166.066,Z 1020.808,A 0.000,B 0.000,C 90.000,E1 145.435} C_DIS
LIN {X -0.003,Y -171.073,Z 1020.789,A 0.000,B 0.000,C 90.000,E1 141.949} C_DIS
LIN {X 0.053,Y -175.946,Z 1020.769,A 0.000,B 0.000,C 90.000,E1 138.485} C_DIS
LIN {X -0.087,Y -180.187,Z 1020.755,A 0.000,B 0.000,C 90.000,E1 135.972} C_DIS
LIN {X -0.119,Y -185.603,Z 1020.737,A 0.000,B 0.000,C 90.000,E1 132.609} C_DIS
LIN {X -0.070,Y -190.196,Z 1020.723,A 0.000,B 0.000,C 90.000,E1 130.092} C_DIS
LIN {X -0.032,Y -196.885,Z 1020.702,A 0.000,B 0.000,C 90.000,E1 126.297} C_DIS
LIN {X -0.102,Y -301.608,Z 1020.702,A 0.000,B 0.000,C 90.000,E1 126.297} C_DIS
LIN {X -0.018,Y -303.610,Z 1020.701,A 0.000,B 0.000,C 90.000,E1 126.251} C_DIS
LIN {X -0.041,Y -309.195,Z 1020.700,A 0.000,B 0.000,C 90.000,E1 125.964} C_DIS
LIN {X -0.046,Y -312.351,Z 1020.698,A 0.000,B 0.000,C 90.000,E1 125.644} C_DIS
LIN {X -0.212,Y -315.954,Z 1020.695,A 0.000,B 0.000,C 90.000,E1 125.105} C_DIS
LIN {X 0.023,Y -317.388,Z 1020.693,A 0.000,B 0.000,C 90.000,E1 124.739} C_DIS
LIN {X -0.024,Y -330.780,Z 1020.672,A 0.000,B 0.000,C 90.000,E1 120.924} C_DIS
